KUKA KRL program: Milling_7_1.src

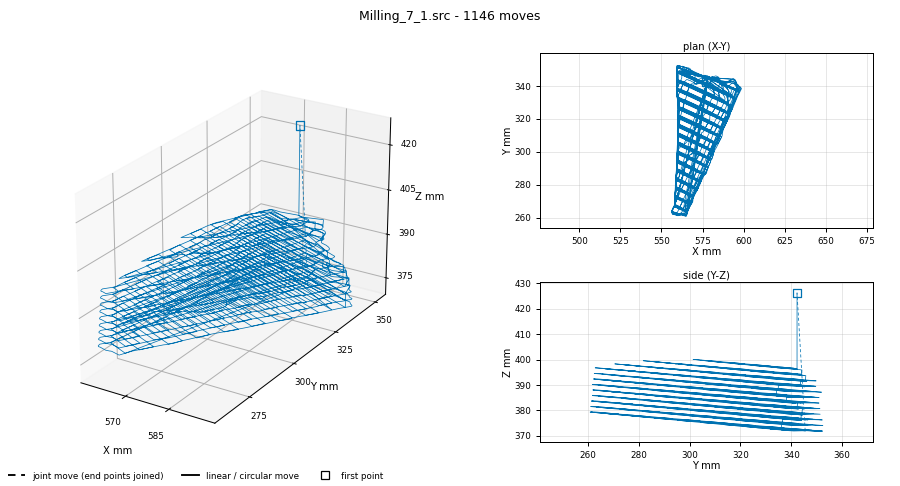
[picture p0: tool path of Milling_7_1.src, 1146 of 1148 moves have a stored position in this frame; points joined in program order, loops and branches not executed]
&ACCESS RVP
&REL 1
&PARAM TEMPLATE = C:\KRC\Roboter\Template\vorgabe
&PARAM EDITMASK = *
DEF Milling_7_1 ( )


;FOLD INI
;FOLD BASISTECH INI
GLOBAL INTERRUPT DECL 3 WHEN $STOPMESS==TRUE DO IR_STOPM ( )
INTERRUPT ON 3
BAS (#INITMOV,0 )
;ENDFOLD (BASISTECH INI)
;ENDFOLD (INI)

;FOLD STARTPOSITION - BASE IS 0, TOOL IS 5, SPEED IS 15%, POSITION IS A1 5,A2 -90,A3 100,A4 5,A5 -10,A6 -5,E1 0,E2 0,E3 0,E4 0
$BWDSTART = FALSE
PDAT_ACT = {VEL 15,ACC 100,APO_DIST 50}
FDAT_ACT = {TOOL_NO 5,BASE_NO 0,IPO_FRAME #BASE}
BAS (#PTP_PARAMS,15)
PTP  {A1 5,A2 -90,A3 100,A4 5,A5 -10,A6 -5,E1 0,E2 0,E3 0,E4 0}
;ENDFOLD

;FOLD LIN SPEED IS 0.1 m/sec, INTERPOLATION SETTINGS IN FOLD
$VEL.CP=0.1
$ADVANCE=3
;ENDFOLD

;FOLD COMMANDS IN FOLD. SELECT EDIT/FOLDS/OPEN ALL FOLDS TO DISPLAY
BAS(#VEL_PTP,2)
PTP {X 576.895, Y 342.279, Z 426.279, A -106.87, B 85.042, C -82.235, E1 0, E2 0, E3 0, E4 0, S 'B010'}
$VEL.CP=0.012
LIN {X 576.895, Y 342.279, Z 396.279, A -106.87, B 85.042, C -82.235, E1 0, E2 0, E3 0, E4 0}
LIN {X 581.744, Y 340.059, Z 396.341, A -106.87, B 85.042, C -82.235, E1 0, E2 0, E3 0, E4 0}
LIN {X 582.117, Y 334.409, Z 396.8, A -106.87, B 85.042, C -82.235, E1 0, E2 0, E3 0, E4 0}
LIN {X 567.684, Y 341.018, Z 396.615, A -106.87, B 85.042, C -82.235, E1 0, E2 0, E3 0, E4 0}
LIN {X 565.563, Y 336.511, Z 397.043, A -106.87, B 85.042, C -82.235, E1 0, E2 0, E3 0, E4 0}
LIN {X 579.527, Y 330.116, Z 397.222, A -106.87, B 85.042, C -82.235, E1 0, E2 0, E3 0, E4 0}
LIN {X 577.52, Y 325.556, Z 397.651, A -106.87, B 85.042, C -82.235, E1 0, E2 0, E3 0, E4 0}
LIN {X 563.782, Y 331.847, Z 397.475, A -106.87, B 85.042, C -82.235, E1 0, E2 0, E3 0, E4 0}
LIN {X 563.044, Y 326.706, Z 397.92, A -106.87, B 85.042, C -82.235, E1 0, E2 0, E3 0, E4 0}
LIN {X 574.933, Y 321.262, Z 398.073, A -106.87, B 85.042, C -82.235, E1 0, E2 0, E3 0, E4 0}
LIN {X 572.822, Y 316.749, Z 398.501, A -106.87, B 85.042, C -82.235, E1 0, E2 0, E3 0, E4 0}
LIN {X 561.971, Y 321.718, Z 398.361, A -106.87, B 85.042, C -82.235, E1 0, E2 0, E3 0, E4 0}
LIN {X 560.617, Y 316.859, Z 398.799, A -106.87, B 85.042, C -82.235, E1 0, E2 0, E3 0, E4 0}
LIN {X 570.047, Y 312.541, Z 398.92, A -106.87, B 85.042, C -82.235, E1 0, E2 0, E3 0, E4 0}
LIN {X 567.602, Y 308.181, Z 399.343, A -106.87, B 85.042, C -82.235, E1 0, E2 0, E3 0, E4 0}
LIN {X 560.515, Y 311.427, Z 399.252, A -106.87, B 85.042, C -82.235, E1 0, E2 0, E3 0, E4 0}
LIN {X 560.232, Y 306.077, Z 399.704, A -106.87, B 85.042, C -82.235, E1 0, E2 0, E3 0, E4 0}
LIN {X 563.648, Y 304.513, Z 399.747, A -106.87, B 85.042, C -82.235, E1 0, E2 0, E3 0, E4 0}
LIN {X 578.662, Y 341.831, Z 396.271, A -106.87, B 85.042, C -82.235, E1 0, E2 0, E3 0, E4 0}
LIN {X 576.305, Y 342.332, Z 396.289, A -106.87, B 85.042, C -82.235, E1 0, E2 0, E3 0, E4 0}
LIN {X 571.991, Y 341.308, Z 396.483, A -106.87, B 85.042, C -82.235, E1 0, E2 0, E3 0, E4 0}
LIN {X 570.835, Y 341.133, Z 396.526, A -106.87, B 85.042, C -82.235, E1 0, E2 0, E3 0, E4 0}
LIN {X 568.535, Y 341.335, Z 396.567, A -106.87, B 85.042, C -82.235, E1 0, E2 0, E3 0, E4 0}
LIN {X 567.853, Y 341.191, Z 396.597, A -106.87, B 85.042, C -82.235, E1 0, E2 0, E3 0, E4 0}
LIN {X 567.158, Y 340.508, Z 396.671, A -106.87, B 85.042, C -82.235, E1 0, E2 0, E3 0, E4 0}
LIN {X 563.05, Y 326.75, Z 397.916, A -106.87, B 85.042, C -82.235, E1 0, E2 0, E3 0, E4 0}
LIN {X 560.877, Y 319.29, Z 398.59, A -106.87, B 85.042, C -82.235, E1 0, E2 0, E3 0, E4 0}
LIN {X 560.632, Y 316.448, Z 398.832, A -106.87, B 85.042, C -82.235, E1 0, E2 0, E3 0, E4 0}
LIN {X 560.608, Y 316.404, Z 398.837, A -106.87, B 85.042, C -82.235, E1 0, E2 0, E3 0, E4 0}
LIN {X 560.617, Y 316.329, Z 398.843, A -106.87, B 85.042, C -82.235, E1 0, E2 0, E3 0, E4 0}
LIN {X 560.448, Y 315.956, Z 398.878, A -106.87, B 85.042, C -82.235, E1 0, E2 0, E3 0, E4 0}
LIN {X 560.332, Y 308.805, Z 399.475, A -106.87, B 85.042, C -82.235, E1 0, E2 0, E3 0, E4 0}
LIN {X 559.954, Y 301.605, Z 400.082, A -106.87, B 85.042, C -82.235, E1 0, E2 0, E3 0, E4 0}
LIN {X 559.952, Y 301.317, Z 400.106, A -106.87, B 85.042, C -82.235, E1 0, E2 0, E3 0, E4 0}
LIN {X 561.639, Y 303.062, Z 399.918, A -106.87, B 85.042, C -82.235, E1 0, E2 0, E3 0, E4 0}
LIN {X 561.767, Y 303.415, Z 399.886, A -106.87, B 85.042, C -82.235, E1 0, E2 0, E3 0, E4 0}
LIN {X 564.546, Y 305.063, Z 399.679, A -106.87, B 85.042, C -82.235, E1 0, E2 0, E3 0, E4 0}
LIN {X 566.478, Y 307.418, Z 399.435, A -106.87, B 85.042, C -82.235, E1 0, E2 0, E3 0, E4 0}
LIN {X 567.57, Y 308.14, Z 399.348, A -106.87, B 85.042, C -82.235, E1 0, E2 0, E3 0, E4 0}
LIN {X 574.106, Y 319.807, Z 398.214, A -106.87, B 85.042, C -82.235, E1 0, E2 0, E3 0, E4 0}
LIN {X 577.01, Y 324.074, Z 397.787, A -106.87, B 85.042, C -82.235, E1 0, E2 0, E3 0, E4 0}
LIN {X 577.887, Y 326.646, Z 397.551, A -106.87, B 85.042, C -82.235, E1 0, E2 0, E3 0, E4 0}
LIN {X 577.83, Y 327.569, Z 397.476, A -106.87, B 85.042, C -82.235, E1 0, E2 0, E3 0, E4 0}
LIN {X 578.067, Y 327.791, Z 397.452, A -106.87, B 85.042, C -82.235, E1 0, E2 0, E3 0, E4 0}
LIN {X 578.437, Y 328.851, Z 397.354, A -106.87, B 85.042, C -82.235, E1 0, E2 0, E3 0, E4 0}
LIN {X 579.308, Y 329.694, Z 397.263, A -106.87, B 85.042, C -82.235, E1 0, E2 0, E3 0, E4 0}
LIN {X 580.616, Y 332.368, Z 397.008, A -106.87, B 85.042, C -82.235, E1 0, E2 0, E3 0, E4 0}
LIN {X 581.829, Y 333.598, Z 396.875, A -106.87, B 85.042, C -82.235, E1 0, E2 0, E3 0, E4 0}
LIN {X 582.26, Y 335.087, Z 396.74, A -106.87, B 85.042, C -82.235, E1 0, E2 0, E3 0, E4 0}
LIN {X 581.267, Y 338.076, Z 396.517, A -106.87, B 85.042, C -82.235, E1 0, E2 0, E3 0, E4 0}
LIN {X 581.747, Y 340.003, Z 396.345, A -106.87, B 85.042, C -82.235, E1 0, E2 0, E3 0, E4 0}
LIN {X 581.733, Y 340.279, Z 396.323, A -106.87, B 85.042, C -82.235, E1 0, E2 0, E3 0, E4 0}
LIN {X 580.797, Y 341.376, Z 396.255, A -106.87, B 85.042, C -82.235, E1 0, E2 0, E3 0, E4 0}
LIN {X 578.662, Y 341.831, Z 396.271, A -106.87, B 85.042, C -82.235, E1 0, E2 0, E3 0, E4 0}
LIN {X 584.625, Y 344.218, Z 395.923, A -106.87, B 85.042, C -82.235, E1 0, E2 0, E3 0, E4 0}
LIN {X 584.571, Y 344.039, Z 393.757, A -106.87, B 85.042, C -82.235, E1 0, E2 0, E3 0, E4 0}
LIN {X 582.705, Y 344.893, Z 393.733, A -106.87, B 85.042, C -82.235, E1 0, E2 0, E3 0, E4 0}
LIN {X 574.324, Y 343.252, Z 394.08, A -106.87, B 85.042, C -82.235, E1 0, E2 0, E3 0, E4 0}
LIN {X 584.3, Y 338.684, Z 394.209, A -106.87, B 85.042, C -82.235, E1 0, E2 0, E3 0, E4 0}
LIN {X 585.153, Y 332.814, Z 394.674, A -106.87, B 85.042, C -82.235, E1 0, E2 0, E3 0, E4 0}
LIN {X 563.874, Y 342.559, Z 394.401, A -106.87, B 85.042, C -82.235, E1 0, E2 0, E3 0, E4 0}
LIN {X 561.643, Y 338.101, Z 394.827, A -106.87, B 85.042, C -82.235, E1 0, E2 0, E3 0, E4 0}
LIN {X 583.515, Y 328.084, Z 395.108, A -106.87, B 85.042, C -82.235, E1 0, E2 0, E3 0, E4 0}
LIN {X 580.918, Y 323.795, Z 395.53, A -106.87, B 85.042, C -82.235, E1 0, E2 0, E3 0, E4 0}
LIN {X 560.439, Y 333.174, Z 395.267, A -106.87, B 85.042, C -82.235, E1 0, E2 0, E3 0, E4 0}
LIN {X 560.554, Y 327.641, Z 395.723, A -106.87, B 85.042, C -82.235, E1 0, E2 0, E3 0, E4 0}
LIN {X 579.074, Y 319.16, Z 395.961, A -106.87, B 85.042, C -82.235, E1 0, E2 0, E3 0, E4 0}
LIN {X 576.813, Y 314.717, Z 396.387, A -106.87, B 85.042, C -82.235, E1 0, E2 0, E3 0, E4 0}
LIN {X 560.377, Y 322.243, Z 396.176, A -106.87, B 85.042, C -82.235, E1 0, E2 0, E3 0, E4 0}
LIN {X 560.494, Y 316.71, Z 396.632, A -106.87, B 85.042, C -82.235, E1 0, E2 0, E3 0, E4 0}
LIN {X 574.212, Y 310.428, Z 396.808, A -106.87, B 85.042, C -82.235, E1 0, E2 0, E3 0, E4 0}
LIN {X 572.498, Y 305.734, Z 397.241, A -106.87, B 85.042, C -82.235, E1 0, E2 0, E3 0, E4 0}
LIN {X 560.46, Y 311.247, Z 397.087, A -106.87, B 85.042, C -82.235, E1 0, E2 0, E3 0, E4 0}
LIN {X 560.177, Y 305.898, Z 397.538, A -106.87, B 85.042, C -82.235, E1 0, E2 0, E3 0, E4 0}
LIN {X 570.719, Y 301.07, Z 397.673, A -106.87, B 85.042, C -82.235, E1 0, E2 0, E3 0, E4 0}
LIN {X 566.667, Y 297.446, Z 398.076, A -106.87, B 85.042, C -82.235, E1 0, E2 0, E3 0, E4 0}
LIN {X 559.925, Y 300.534, Z 397.989, A -106.87, B 85.042, C -82.235, E1 0, E2 0, E3 0, E4 0}
LIN {X 560.131, Y 294.96, Z 398.447, A -106.87, B 85.042, C -82.235, E1 0, E2 0, E3 0, E4 0}
LIN {X 563.737, Y 293.309, Z 398.493, A -106.87, B 85.042, C -82.235, E1 0, E2 0, E3 0, E4 0}
LIN {X 562.482, Y 288.404, Z 398.932, A -106.87, B 85.042, C -82.235, E1 0, E2 0, E3 0, E4 0}
LIN {X 559.719, Y 289.67, Z 398.896, A -106.87, B 85.042, C -82.235, E1 0, E2 0, E3 0, E4 0}
LIN {X 559.06, Y 284.492, Z 399.343, A -106.87, B 85.042, C -82.235, E1 0, E2 0, E3 0, E4 0}
LIN {X 560.33, Y 283.911, Z 399.359, A -106.87, B 85.042, C -82.235, E1 0, E2 0, E3 0, E4 0}
LIN {X 578.097, Y 344.003, Z 393.923, A -106.87, B 85.042, C -82.235, E1 0, E2 0, E3 0, E4 0}
LIN {X 583.583, Y 345.174, Z 393.688, A -106.87, B 85.042, C -82.235, E1 0, E2 0, E3 0, E4 0}
LIN {X 583.658, Y 345.166, Z 393.687, A -106.87, B 85.042, C -82.235, E1 0, E2 0, E3 0, E4 0}
LIN {X 583.724, Y 345.117, Z 393.689, A -106.87, B 85.042, C -82.235, E1 0, E2 0, E3 0, E4 0}
LIN {X 585.069, Y 343.343, Z 393.802, A -106.87, B 85.042, C -82.235, E1 0, E2 0, E3 0, E4 0}
LIN {X 585.534, Y 341.633, Z 393.933, A -106.87, B 85.042, C -82.235, E1 0, E2 0, E3 0, E4 0}
LIN {X 585.454, Y 341.123, Z 393.977, A -106.87, B 85.042, C -82.235, E1 0, E2 0, E3 0, E4 0}
LIN {X 584.65, Y 339.762, Z 394.11, A -106.87, B 85.042, C -82.235, E1 0, E2 0, E3 0, E4 0}
LIN {X 584.558, Y 339.684, Z 394.119, A -106.87, B 85.042, C -82.235, E1 0, E2 0, E3 0, E4 0}
LIN {X 584.115, Y 337.478, Z 394.313, A -106.87, B 85.042, C -82.235, E1 0, E2 0, E3 0, E4 0}
LIN {X 585.114, Y 335.114, Z 394.484, A -106.87, B 85.042, C -82.235, E1 0, E2 0, E3 0, E4 0}
LIN {X 585.144, Y 332.703, Z 394.684, A -106.87, B 85.042, C -82.235, E1 0, E2 0, E3 0, E4 0}
LIN {X 584.551, Y 331.291, Z 394.816, A -106.87, B 85.042, C -82.235, E1 0, E2 0, E3 0, E4 0}
LIN {X 584.057, Y 330.694, Z 394.878, A -106.87, B 85.042, C -82.235, E1 0, E2 0, E3 0, E4 0}
LIN {X 583.581, Y 328.244, Z 395.093, A -106.87, B 85.042, C -82.235, E1 0, E2 0, E3 0, E4 0}
LIN {X 580.825, Y 323.667, Z 395.543, A -106.87, B 85.042, C -82.235, E1 0, E2 0, E3 0, E4 0}
LIN {X 579.822, Y 323.235, Z 395.604, A -106.87, B 85.042, C -82.235, E1 0, E2 0, E3 0, E4 0}
LIN {X 579.732, Y 323.124, Z 395.615, A -106.87, B 85.042, C -82.235, E1 0, E2 0, E3 0, E4 0}
LIN {X 579.441, Y 322.375, Z 395.685, A -106.87, B 85.042, C -82.235, E1 0, E2 0, E3 0, E4 0}
LIN {X 579.352, Y 319.987, Z 395.885, A -106.87, B 85.042, C -82.235, E1 0, E2 0, E3 0, E4 0}
LIN {X 576.924, Y 315.102, Z 396.352, A -106.87, B 85.042, C -82.235, E1 0, E2 0, E3 0, E4 0}
LIN {X 576.416, Y 313.428, Z 396.504, A -106.87, B 85.042, C -82.235, E1 0, E2 0, E3 0, E4 0}
LIN {X 575.142, Y 311.958, Z 396.658, A -106.87, B 85.042, C -82.235, E1 0, E2 0, E3 0, E4 0}
LIN {X 574.554, Y 311.675, Z 396.696, A -106.87, B 85.042, C -82.235, E1 0, E2 0, E3 0, E4 0}
LIN {X 574.252, Y 311.233, Z 396.74, A -106.87, B 85.042, C -82.235, E1 0, E2 0, E3 0, E4 0}
LIN {X 574.21, Y 309.999, Z 396.844, A -106.87, B 85.042, C -82.235, E1 0, E2 0, E3 0, E4 0}
LIN {X 570.659, Y 300.834, Z 397.694, A -106.87, B 85.042, C -82.235, E1 0, E2 0, E3 0, E4 0}
LIN {X 569.22, Y 298.941, Z 397.888, A -106.87, B 85.042, C -82.235, E1 0, E2 0, E3 0, E4 0}
LIN {X 566.753, Y 297.93, Z 398.034, A -106.87, B 85.042, C -82.235, E1 0, E2 0, E3 0, E4 0}
LIN {X 566.692, Y 297.837, Z 398.043, A -106.87, B 85.042, C -82.235, E1 0, E2 0, E3 0, E4 0}
LIN {X 566.762, Y 296.23, Z 398.175, A -106.87, B 85.042, C -82.235, E1 0, E2 0, E3 0, E4 0}
LIN {X 566.431, Y 295.493, Z 398.244, A -106.87, B 85.042, C -82.235, E1 0, E2 0, E3 0, E4 0}
LIN {X 566.28, Y 294.839, Z 398.302, A -106.87, B 85.042, C -82.235, E1 0, E2 0, E3 0, E4 0}
LIN {X 565.783, Y 294.409, Z 398.35, A -106.87, B 85.042, C -82.235, E1 0, E2 0, E3 0, E4 0}
LIN {X 565.156, Y 294.696, Z 398.342, A -106.87, B 85.042, C -82.235, E1 0, E2 0, E3 0, E4 0}
LIN {X 564.945, Y 294.236, Z 398.386, A -106.87, B 85.042, C -82.235, E1 0, E2 0, E3 0, E4 0}
LIN {X 564.12, Y 293.972, Z 398.429, A -106.87, B 85.042, C -82.235, E1 0, E2 0, E3 0, E4 0}
LIN {X 563.85, Y 293.432, Z 398.48, A -106.87, B 85.042, C -82.235, E1 0, E2 0, E3 0, E4 0}
LIN {X 563.685, Y 293.251, Z 398.499, A -106.87, B 85.042, C -82.235, E1 0, E2 0, E3 0, E4 0}
LIN {X 564.591, Y 292.757, Z 398.518, A -106.87, B 85.042, C -82.235, E1 0, E2 0, E3 0, E4 0}
LIN {X 564.637, Y 292.748, Z 398.517, A -106.87, B 85.042, C -82.235, E1 0, E2 0, E3 0, E4 0}
LIN {X 564.633, Y 292.727, Z 398.519, A -106.87, B 85.042, C -82.235, E1 0, E2 0, E3 0, E4 0}
LIN {X 564.76, Y 291.881, Z 398.586, A -106.87, B 85.042, C -82.235, E1 0, E2 0, E3 0, E4 0}
LIN {X 564.136, Y 290.632, Z 398.705, A -106.87, B 85.042, C -82.235, E1 0, E2 0, E3 0, E4 0}
LIN {X 563.633, Y 290.496, Z 398.729, A -106.87, B 85.042, C -82.235, E1 0, E2 0, E3 0, E4 0}
LIN {X 563.816, Y 290.033, Z 398.763, A -106.87, B 85.042, C -82.235, E1 0, E2 0, E3 0, E4 0}
LIN {X 562.653, Y 288.496, Z 398.92, A -106.87, B 85.042, C -82.235, E1 0, E2 0, E3 0, E4 0}
LIN {X 562.089, Y 288.191, Z 398.96, A -106.87, B 85.042, C -82.235, E1 0, E2 0, E3 0, E4 0}
LIN {X 561.588, Y 287.183, Z 399.056, A -106.87, B 85.042, C -82.235, E1 0, E2 0, E3 0, E4 0}
LIN {X 561.726, Y 286.954, Z 399.071, A -106.87, B 85.042, C -82.235, E1 0, E2 0, E3 0, E4 0}
LIN {X 561.239, Y 286.678, Z 399.107, A -106.87, B 85.042, C -82.235, E1 0, E2 0, E3 0, E4 0}
LIN {X 561.257, Y 286.467, Z 399.124, A -106.87, B 85.042, C -82.235, E1 0, E2 0, E3 0, E4 0}
LIN {X 560.71, Y 284.65, Z 399.288, A -106.87, B 85.042, C -82.235, E1 0, E2 0, E3 0, E4 0}
LIN {X 559.03, Y 281.698, Z 399.576, A -106.87, B 85.042, C -82.235, E1 0, E2 0, E3 0, E4 0}
LIN {X 560.519, Y 309.67, Z 397.216, A -106.87, B 85.042, C -82.235, E1 0, E2 0, E3 0, E4 0}
LIN {X 560.165, Y 314.552, Z 396.82, A -106.87, B 85.042, C -82.235, E1 0, E2 0, E3 0, E4 0}
LIN {X 560.562, Y 316.149, Z 396.677, A -106.87, B 85.042, C -82.235, E1 0, E2 0, E3 0, E4 0}
LIN {X 560.48, Y 317.178, Z 396.594, A -106.87, B 85.042, C -82.235, E1 0, E2 0, E3 0, E4 0}
LIN {X 560.446, Y 317.247, Z 396.589, A -106.87, B 85.042, C -82.235, E1 0, E2 0, E3 0, E4 0}
LIN {X 560.814, Y 330.69, Z 395.464, A -106.87, B 85.042, C -82.235, E1 0, E2 0, E3 0, E4 0}
LIN {X 560.738, Y 330.851, Z 395.452, A -106.87, B 85.042, C -82.235, E1 0, E2 0, E3 0, E4 0}
LIN {X 560.306, Y 334.39, Z 395.169, A -106.87, B 85.042, C -82.235, E1 0, E2 0, E3 0, E4 0}
LIN {X 563.334, Y 341.786, Z 394.479, A -106.87, B 85.042, C -82.235, E1 0, E2 0, E3 0, E4 0}
LIN {X 565.199, Y 343.887, Z 394.257, A -106.87, B 85.042, C -82.235, E1 0, E2 0, E3 0, E4 0}
LIN {X 566.09, Y 343.841, Z 394.239, A -106.87, B 85.042, C -82.235, E1 0, E2 0, E3 0, E4 0}
LIN {X 566.53, Y 343.532, Z 394.253, A -106.87, B 85.042, C -82.235, E1 0, E2 0, E3 0, E4 0}
LIN {X 567.45, Y 343.318, Z 394.248, A -106.87, B 85.042, C -82.235, E1 0, E2 0, E3 0, E4 0}
LIN {X 570.821, Y 341.414, Z 394.321, A -106.87, B 85.042, C -82.235, E1 0, E2 0, E3 0, E4 0}
LIN {X 571.518, Y 341.33, Z 394.311, A -106.87, B 85.042, C -82.235, E1 0, E2 0, E3 0, E4 0}
LIN {X 573.337, Y 342.631, Z 394.157, A -106.87, B 85.042, C -82.235, E1 0, E2 0, E3 0, E4 0}
LIN {X 573.683, Y 343.06, Z 394.112, A -106.87, B 85.042, C -82.235, E1 0, E2 0, E3 0, E4 0}
LIN {X 578.097, Y 344.003, Z 393.923, A -106.87, B 85.042, C -82.235, E1 0, E2 0, E3 0, E4 0}
LIN {X 580.876, Y 345.731, Z 393.71, A -106.87, B 85.042, C -82.235, E1 0, E2 0, E3 0, E4 0}
LIN {X 580.822, Y 345.551, Z 391.544, A -106.87, B 85.042, C -82.235, E1 0, E2 0, E3 0, E4 0}
LIN {X 585.842, Y 343.252, Z 391.608, A -106.87, B 85.042, C -82.235, E1 0, E2 0, E3 0, E4 0}
LIN {X 587.33, Y 337.091, Z 392.082, A -106.87, B 85.042, C -82.235, E1 0, E2 0, E3 0, E4 0}
LIN {X 572.399, Y 343.929, Z 391.891, A -106.87, B 85.042, C -82.235, E1 0, E2 0, E3 0, E4 0}
LIN {X 562.627, Y 348.404, Z 391.765, A -106.87, B 85.042, C -82.235, E1 0, E2 0, E3 0, E4 0}
LIN {X 570.487, Y 344.804, Z 391.866, A -106.87, B 85.042, C -82.235, E1 0, E2 0, E3 0, E4 0}
LIN {X 588.468, Y 331.091, Z 392.552, A -106.87, B 85.042, C -82.235, E1 0, E2 0, E3 0, E4 0}
LIN {X 561.576, Y 343.406, Z 392.207, A -106.87, B 85.042, C -82.235, E1 0, E2 0, E3 0, E4 0}
LIN {X 559.643, Y 338.812, Z 392.637, A -106.87, B 85.042, C -82.235, E1 0, E2 0, E3 0, E4 0}
LIN {X 586.399, Y 326.559, Z 392.98, A -106.87, B 85.042, C -82.235, E1 0, E2 0, E3 0, E4 0}
LIN {X 584.074, Y 322.145, Z 393.405, A -106.87, B 85.042, C -82.235, E1 0, E2 0, E3 0, E4 0}
LIN {X 560.384, Y 332.994, Z 393.101, A -106.87, B 85.042, C -82.235, E1 0, E2 0, E3 0, E4 0}
LIN {X 560.5, Y 327.462, Z 393.557, A -106.87, B 85.042, C -82.235, E1 0, E2 0, E3 0, E4 0}
LIN {X 581.809, Y 317.703, Z 393.831, A -106.87, B 85.042, C -82.235, E1 0, E2 0, E3 0, E4 0}
LIN {X 579.849, Y 313.121, Z 394.261, A -106.87, B 85.042, C -82.235, E1 0, E2 0, E3 0, E4 0}
LIN {X 560.323, Y 322.063, Z 394.01, A -106.87, B 85.042, C -82.235, E1 0, E2 0, E3 0, E4 0}
LIN {X 560.44, Y 316.531, Z 394.466, A -106.87, B 85.042, C -82.235, E1 0, E2 0, E3 0, E4 0}
LIN {X 577.836, Y 308.564, Z 394.69, A -106.87, B 85.042, C -82.235, E1 0, E2 0, E3 0, E4 0}
LIN {X 575.845, Y 303.996, Z 395.119, A -106.87, B 85.042, C -82.235, E1 0, E2 0, E3 0, E4 0}
LIN {X 560.406, Y 311.067, Z 394.921, A -106.87, B 85.042, C -82.235, E1 0, E2 0, E3 0, E4 0}
LIN {X 560.122, Y 305.718, Z 395.372, A -106.87, B 85.042, C -82.235, E1 0, E2 0, E3 0, E4 0}
LIN {X 573.777, Y 299.464, Z 395.547, A -106.87, B 85.042, C -82.235, E1 0, E2 0, E3 0, E4 0}
LIN {X 571.315, Y 295.113, Z 395.971, A -106.87, B 85.042, C -82.235, E1 0, E2 0, E3 0, E4 0}
LIN {X 559.871, Y 300.354, Z 395.824, A -106.87, B 85.042, C -82.235, E1 0, E2 0, E3 0, E4 0}
LIN {X 560.076, Y 294.781, Z 396.281, A -106.87, B 85.042, C -82.235, E1 0, E2 0, E3 0, E4 0}
LIN {X 569.346, Y 290.535, Z 396.4, A -106.87, B 85.042, C -82.235, E1 0, E2 0, E3 0, E4 0}
LIN {X 566.96, Y 286.149, Z 396.824, A -106.87, B 85.042, C -82.235, E1 0, E2 0, E3 0, E4 0}
LIN {X 559.664, Y 289.49, Z 396.731, A -106.87, B 85.042, C -82.235, E1 0, E2 0, E3 0, E4 0}
LIN {X 559.006, Y 284.312, Z 397.177, A -106.87, B 85.042, C -82.235, E1 0, E2 0, E3 0, E4 0}
LIN {X 564.493, Y 281.799, Z 397.248, A -106.87, B 85.042, C -82.235, E1 0, E2 0, E3 0, E4 0}
LIN {X 562.21, Y 277.366, Z 397.673, A -106.87, B 85.042, C -82.235, E1 0, E2 0, E3 0, E4 0}
LIN {X 558.844, Y 278.907, Z 397.63, A -106.87, B 85.042, C -82.235, E1 0, E2 0, E3 0, E4 0}
LIN {X 558.518, Y 273.577, Z 398.081, A -106.87, B 85.042, C -82.235, E1 0, E2 0, E3 0, E4 0}
LIN {X 559.993, Y 272.902, Z 398.1, A -106.87, B 85.042, C -82.235, E1 0, E2 0, E3 0, E4 0}
LIN {X 578.218, Y 345.098, Z 391.647, A -106.87, B 85.042, C -82.235, E1 0, E2 0, E3 0, E4 0}
LIN {X 579.101, Y 344.975, Z 391.635, A -106.87, B 85.042, C -82.235, E1 0, E2 0, E3 0, E4 0}
LIN {X 583.083, Y 346.167, Z 391.436, A -106.87, B 85.042, C -82.235, E1 0, E2 0, E3 0, E4 0}
LIN {X 584.478, Y 345.556, Z 391.451, A -106.87, B 85.042, C -82.235, E1 0, E2 0, E3 0, E4 0}
LIN {X 585.511, Y 344.183, Z 391.539, A -106.87, B 85.042, C -82.235, E1 0, E2 0, E3 0, E4 0}
LIN {X 586.277, Y 340.991, Z 391.785, A -106.87, B 85.042, C -82.235, E1 0, E2 0, E3 0, E4 0}
LIN {X 587.074, Y 340.037, Z 391.844, A -106.87, B 85.042, C -82.235, E1 0, E2 0, E3 0, E4 0}
LIN {X 587.651, Y 339.495, Z 391.875, A -106.87, B 85.042, C -82.235, E1 0, E2 0, E3 0, E4 0}
LIN {X 587.856, Y 338.588, Z 391.945, A -106.87, B 85.042, C -82.235, E1 0, E2 0, E3 0, E4 0}
LIN {X 587.296, Y 336.993, Z 392.091, A -106.87, B 85.042, C -82.235, E1 0, E2 0, E3 0, E4 0}
LIN {X 587.229, Y 335.812, Z 392.191, A -106.87, B 85.042, C -82.235, E1 0, E2 0, E3 0, E4 0}
LIN {X 587.483, Y 334.662, Z 392.28, A -106.87, B 85.042, C -82.235, E1 0, E2 0, E3 0, E4 0}
LIN {X 588.142, Y 333.798, Z 392.335, A -106.87, B 85.042, C -82.235, E1 0, E2 0, E3 0, E4 0}
LIN {X 588.645, Y 332.542, Z 392.427, A -106.87, B 85.042, C -82.235, E1 0, E2 0, E3 0, E4 0}
LIN {X 588.395, Y 330.692, Z 392.587, A -106.87, B 85.042, C -82.235, E1 0, E2 0, E3 0, E4 0}
LIN {X 581.012, Y 315.463, Z 394.037, A -106.87, B 85.042, C -82.235, E1 0, E2 0, E3 0, E4 0}
LIN {X 561.669, Y 276.539, Z 397.755, A -106.87, B 85.042, C -82.235, E1 0, E2 0, E3 0, E4 0}
LIN {X 561.673, Y 276.429, Z 397.764, A -106.87, B 85.042, C -82.235, E1 0, E2 0, E3 0, E4 0}
LIN {X 560.774, Y 274.04, Z 397.986, A -106.87, B 85.042, C -82.235, E1 0, E2 0, E3 0, E4 0}
LIN {X 558.721, Y 270.49, Z 398.332, A -106.87, B 85.042, C -82.235, E1 0, E2 0, E3 0, E4 0}
LIN {X 558.537, Y 272.628, Z 398.159, A -106.87, B 85.042, C -82.235, E1 0, E2 0, E3 0, E4 0}
LIN {X 558.828, Y 276.652, Z 397.818, A -106.87, B 85.042, C -82.235, E1 0, E2 0, E3 0, E4 0}
LIN {X 560.465, Y 309.49, Z 395.05, A -106.87, B 85.042, C -82.235, E1 0, E2 0, E3 0, E4 0}
LIN {X 560.11, Y 314.372, Z 394.654, A -106.87, B 85.042, C -82.235, E1 0, E2 0, E3 0, E4 0}
LIN {X 560.508, Y 315.969, Z 394.511, A -106.87, B 85.042, C -82.235, E1 0, E2 0, E3 0, E4 0}
LIN {X 560.425, Y 316.998, Z 394.428, A -106.87, B 85.042, C -82.235, E1 0, E2 0, E3 0, E4 0}
LIN {X 560.391, Y 317.067, Z 394.423, A -106.87, B 85.042, C -82.235, E1 0, E2 0, E3 0, E4 0}
LIN {X 560.759, Y 330.511, Z 393.298, A -106.87, B 85.042, C -82.235, E1 0, E2 0, E3 0, E4 0}
LIN {X 560.683, Y 330.671, Z 393.286, A -106.87, B 85.042, C -82.235, E1 0, E2 0, E3 0, E4 0}
LIN {X 559.737, Y 335.976, Z 392.87, A -106.87, B 85.042, C -82.235, E1 0, E2 0, E3 0, E4 0}
LIN {X 559.647, Y 339.062, Z 392.616, A -106.87, B 85.042, C -82.235, E1 0, E2 0, E3 0, E4 0}
LIN {X 562.296, Y 344.753, Z 392.077, A -106.87, B 85.042, C -82.235, E1 0, E2 0, E3 0, E4 0}
LIN {X 562.552, Y 349.38, Z 391.686, A -106.87, B 85.042, C -82.235, E1 0, E2 0, E3 0, E4 0}
LIN {X 562.628, Y 349.761, Z 391.652, A -106.87, B 85.042, C -82.235, E1 0, E2 0, E3 0, E4 0}
LIN {X 562.694, Y 349.794, Z 391.648, A -106.87, B 85.042, C -82.235, E1 0, E2 0, E3 0, E4 0}
LIN {X 566.596, Y 348.974, Z 391.618, A -106.87, B 85.042, C -82.235, E1 0, E2 0, E3 0, E4 0}
LIN {X 569.925, Y 347.68, Z 391.641, A -106.87, B 85.042, C -82.235, E1 0, E2 0, E3 0, E4 0}
LIN {X 570.226, Y 347.271, Z 391.668, A -106.87, B 85.042, C -82.235, E1 0, E2 0, E3 0, E4 0}
LIN {X 570.209, Y 347.141, Z 391.679, A -106.87, B 85.042, C -82.235, E1 0, E2 0, E3 0, E4 0}
LIN {X 570.438, Y 346.095, Z 391.76, A -106.87, B 85.042, C -82.235, E1 0, E2 0, E3 0, E4 0}
LIN {X 570.351, Y 344.929, Z 391.859, A -106.87, B 85.042, C -82.235, E1 0, E2 0, E3 0, E4 0}
LIN {X 571.715, Y 343.685, Z 391.928, A -106.87, B 85.042, C -82.235, E1 0, E2 0, E3 0, E4 0}
LIN {X 569.859, Y 343.017, Z 392.03, A -106.87, B 85.042, C -82.235, E1 0, E2 0, E3 0, E4 0}
LIN {X 569.861, Y 342.66, Z 392.06, A -106.87, B 85.042, C -82.235, E1 0, E2 0, E3 0, E4 0}
LIN {X 569.65, Y 342.247, Z 392.099, A -106.87, B 85.042, C -82.235, E1 0, E2 0, E3 0, E4 0}
LIN {X 570.082, Y 341.636, Z 392.139, A -106.87, B 85.042, C -82.235, E1 0, E2 0, E3 0, E4 0}
LIN {X 570.349, Y 341.468, Z 392.147, A -106.87, B 85.042, C -82.235, E1 0, E2 0, E3 0, E4 0}
LIN {X 571.203, Y 341.242, Z 392.144, A -106.87, B 85.042, C -82.235, E1 0, E2 0, E3 0, E4 0}
LIN {X 571.783, Y 343.654, Z 391.929, A -106.87, B 85.042, C -82.235, E1 0, E2 0, E3 0, E4 0}
LIN {X 571.795, Y 343.669, Z 391.927, A -106.87, B 85.042, C -82.235, E1 0, E2 0, E3 0, E4 0}
LIN {X 574.195, Y 344.701, Z 391.781, A -106.87, B 85.042, C -82.235, E1 0, E2 0, E3 0, E4 0}
LIN {X 576.649, Y 344.932, Z 391.7, A -106.87, B 85.042, C -82.235, E1 0, E2 0, E3 0, E4 0}
LIN {X 577.654, Y 345.176, Z 391.655, A -106.87, B 85.042, C -82.235, E1 0, E2 0, E3 0, E4 0}
LIN {X 578.218, Y 345.098, Z 391.647, A -106.87, B 85.042, C -82.235, E1 0, E2 0, E3 0, E4 0}
LIN {X 584.892, Y 343.687, Z 391.596, A -106.87, B 85.042, C -82.235, E1 0, E2 0, E3 0, E4 0}
LIN {X 584.837, Y 343.507, Z 389.43, A -106.87, B 85.042, C -82.235, E1 0, E2 0, E3 0, E4 0}
LIN {X 581.654, Y 344.965, Z 389.389, A -106.87, B 85.042, C -82.235, E1 0, E2 0, E3 0, E4 0}
LIN {X 560.751, Y 349.059, Z 389.576, A -106.87, B 85.042, C -82.235, E1 0, E2 0, E3 0, E4 0}
LIN {X 590.147, Y 335.596, Z 389.954, A -106.87, B 85.042, C -82.235, E1 0, E2 0, E3 0, E4 0}
LIN {X 590.276, Y 330.058, Z 390.41, A -106.87, B 85.042, C -82.235, E1 0, E2 0, E3 0, E4 0}
LIN {X 559.646, Y 344.085, Z 390.017, A -106.87, B 85.042, C -82.235, E1 0, E2 0, E3 0, E4 0}
LIN {X 559.589, Y 338.633, Z 390.471, A -106.87, B 85.042, C -82.235, E1 0, E2 0, E3 0, E4 0}
LIN {X 588.617, Y 325.339, Z 390.844, A -106.87, B 85.042, C -82.235, E1 0, E2 0, E3 0, E4 0}
LIN {X 586.307, Y 320.917, Z 391.269, A -106.87, B 85.042, C -82.235, E1 0, E2 0, E3 0, E4 0}
LIN {X 560.33, Y 332.814, Z 390.935, A -106.87, B 85.042, C -82.235, E1 0, E2 0, E3 0, E4 0}
LIN {X 560.445, Y 327.282, Z 391.392, A -106.87, B 85.042, C -82.235, E1 0, E2 0, E3 0, E4 0}
LIN {X 584.357, Y 316.331, Z 391.699, A -106.87, B 85.042, C -82.235, E1 0, E2 0, E3 0, E4 0}
LIN {X 582.293, Y 311.797, Z 392.127, A -106.87, B 85.042, C -82.235, E1 0, E2 0, E3 0, E4 0}
LIN {X 560.268, Y 321.884, Z 391.844, A -106.87, B 85.042, C -82.235, E1 0, E2 0, E3 0, E4 0}
LIN {X 560.385, Y 316.351, Z 392.301, A -106.87, B 85.042, C -82.235, E1 0, E2 0, E3 0, E4 0}
LIN {X 580.214, Y 307.27, Z 392.555, A -106.87, B 85.042, C -82.235, E1 0, E2 0, E3 0, E4 0}
LIN {X 578.281, Y 302.676, Z 392.985, A -106.87, B 85.042, C -82.235, E1 0, E2 0, E3 0, E4 0}
LIN {X 560.351, Y 310.887, Z 392.755, A -106.87, B 85.042, C -82.235, E1 0, E2 0, E3 0, E4 0}
LIN {X 560.068, Y 305.538, Z 393.206, A -106.87, B 85.042, C -82.235, E1 0, E2 0, E3 0, E4 0}
LIN {X 576.165, Y 298.166, Z 393.413, A -106.87, B 85.042, C -82.235, E1 0, E2 0, E3 0, E4 0}
LIN {X 574.194, Y 293.59, Z 393.842, A -106.87, B 85.042, C -82.235, E1 0, E2 0, E3 0, E4 0}
LIN {X 559.816, Y 300.174, Z 393.658, A -106.87, B 85.042, C -82.235, E1 0, E2 0, E3 0, E4 0}
LIN {X 560.022, Y 294.601, Z 394.115, A -106.87, B 85.042, C -82.235, E1 0, E2 0, E3 0, E4 0}
LIN {X 572.043, Y 289.096, Z 394.27, A -106.87, B 85.042, C -82.235, E1 0, E2 0, E3 0, E4 0}
LIN {X 569.847, Y 284.622, Z 394.696, A -106.87, B 85.042, C -82.235, E1 0, E2 0, E3 0, E4 0}
LIN {X 559.609, Y 289.31, Z 394.565, A -106.87, B 85.042, C -82.235, E1 0, E2 0, E3 0, E4 0}
LIN {X 558.951, Y 284.133, Z 395.011, A -106.87, B 85.042, C -82.235, E1 0, E2 0, E3 0, E4 0}
LIN {X 568.041, Y 279.97, Z 395.128, A -106.87, B 85.042, C -82.235, E1 0, E2 0, E3 0, E4 0}
LIN {X 565.556, Y 275.628, Z 395.551, A -106.87, B 85.042, C -82.235, E1 0, E2 0, E3 0, E4 0}
LIN {X 558.789, Y 278.728, Z 395.464, A -106.87, B 85.042, C -82.235, E1 0, E2 0, E3 0, E4 0}
LIN {X 558.463, Y 273.398, Z 395.915, A -106.87, B 85.042, C -82.235, E1 0, E2 0, E3 0, E4 0}
LIN {X 563.541, Y 271.072, Z 395.98, A -106.87, B 85.042, C -82.235, E1 0, E2 0, E3 0, E4 0}
LIN {X 561.262, Y 266.637, Z 396.406, A -106.87, B 85.042, C -82.235, E1 0, E2 0, E3 0, E4 0}
LIN {X 558.324, Y 267.982, Z 396.368, A -106.87, B 85.042, C -82.235, E1 0, E2 0, E3 0, E4 0}
LIN {X 578.154, Y 344.821, Z 389.49, A -106.87, B 85.042, C -82.235, E1 0, E2 0, E3 0, E4 0}
LIN {X 580.331, Y 344.607, Z 389.453, A -106.87, B 85.042, C -82.235, E1 0, E2 0, E3 0, E4 0}
LIN {X 583.657, Y 345.363, Z 389.306, A -106.87, B 85.042, C -82.235, E1 0, E2 0, E3 0, E4 0}
LIN {X 584.034, Y 345.169, Z 389.313, A -106.87, B 85.042, C -82.235, E1 0, E2 0, E3 0, E4 0}
LIN {X 585.184, Y 342.399, Z 389.514, A -106.87, B 85.042, C -82.235, E1 0, E2 0, E3 0, E4 0}
LIN {X 585.762, Y 341.122, Z 389.605, A -106.87, B 85.042, C -82.235, E1 0, E2 0, E3 0, E4 0}
LIN {X 586.211, Y 340.748, Z 389.625, A -106.87, B 85.042, C -82.235, E1 0, E2 0, E3 0, E4 0}
LIN {X 588.162, Y 340.013, Z 389.637, A -106.87, B 85.042, C -82.235, E1 0, E2 0, E3 0, E4 0}
LIN {X 589.656, Y 338.99, Z 389.684, A -106.87, B 85.042, C -82.235, E1 0, E2 0, E3 0, E4 0}
LIN {X 590.535, Y 337.925, Z 389.75, A -106.87, B 85.042, C -82.235, E1 0, E2 0, E3 0, E4 0}
LIN {X 590.85, Y 336.932, Z 389.825, A -106.87, B 85.042, C -82.235, E1 0, E2 0, E3 0, E4 0}
LIN {X 590.748, Y 336.368, Z 389.874, A -106.87, B 85.042, C -82.235, E1 0, E2 0, E3 0, E4 0}
LIN {X 590.588, Y 336.043, Z 389.905, A -106.87, B 85.042, C -82.235, E1 0, E2 0, E3 0, E4 0}
LIN {X 589.712, Y 335.082, Z 390.007, A -106.87, B 85.042, C -82.235, E1 0, E2 0, E3 0, E4 0}
LIN {X 589.573, Y 333.596, Z 390.134, A -106.87, B 85.042, C -82.235, E1 0, E2 0, E3 0, E4 0}
LIN {X 590.534, Y 331.255, Z 390.304, A -106.87, B 85.042, C -82.235, E1 0, E2 0, E3 0, E4 0}
LIN {X 590.525, Y 331.073, Z 390.319, A -106.87, B 85.042, C -82.235, E1 0, E2 0, E3 0, E4 0}
LIN {X 589.274, Y 327.373, Z 390.658, A -106.87, B 85.042, C -82.235, E1 0, E2 0, E3 0, E4 0}
LIN {X 589.277, Y 327.253, Z 390.668, A -106.87, B 85.042, C -82.235, E1 0, E2 0, E3 0, E4 0}
LIN {X 586.482, Y 321.496, Z 391.216, A -106.87, B 85.042, C -82.235, E1 0, E2 0, E3 0, E4 0}
LIN {X 585.884, Y 319.472, Z 391.399, A -106.87, B 85.042, C -82.235, E1 0, E2 0, E3 0, E4 0}
LIN {X 584.756, Y 317.738, Z 391.572, A -106.87, B 85.042, C -82.235, E1 0, E2 0, E3 0, E4 0}
LIN {X 560.637, Y 265.269, Z 396.535, A -106.87, B 85.042, C -82.235, E1 0, E2 0, E3 0, E4 0}
LIN {X 559.469, Y 262.754, Z 396.773, A -106.87, B 85.042, C -82.235, E1 0, E2 0, E3 0, E4 0}
LIN {X 557.985, Y 263.322, Z 396.763, A -106.87, B 85.042, C -82.235, E1 0, E2 0, E3 0, E4 0}
LIN {X 557.364, Y 263.333, Z 396.778, A -106.87, B 85.042, C -82.235, E1 0, E2 0, E3 0, E4 0}
LIN {X 556.928, Y 263.837, Z 396.747, A -106.87, B 85.042, C -82.235, E1 0, E2 0, E3 0, E4 0}
LIN {X 556.637, Y 265.071, Z 396.652, A -106.87, B 85.042, C -82.235, E1 0, E2 0, E3 0, E4 0}
LIN {X 558.536, Y 268.72, Z 396.302, A -106.87, B 85.042, C -82.235, E1 0, E2 0, E3 0, E4 0}
LIN {X 558.483, Y 272.448, Z 395.993, A -106.87, B 85.042, C -82.235, E1 0, E2 0, E3 0, E4 0}
LIN {X 558.774, Y 276.473, Z 395.652, A -106.87, B 85.042, C -82.235, E1 0, E2 0, E3 0, E4 0}
LIN {X 560.41, Y 309.31, Z 392.885, A -106.87, B 85.042, C -82.235, E1 0, E2 0, E3 0, E4 0}
LIN {X 560.056, Y 314.193, Z 392.488, A -106.87, B 85.042, C -82.235, E1 0, E2 0, E3 0, E4 0}
LIN {X 560.453, Y 315.79, Z 392.345, A -106.87, B 85.042, C -82.235, E1 0, E2 0, E3 0, E4 0}
LIN {X 560.371, Y 316.818, Z 392.262, A -106.87, B 85.042, C -82.235, E1 0, E2 0, E3 0, E4 0}
LIN {X 560.337, Y 316.887, Z 392.257, A -106.87, B 85.042, C -82.235, E1 0, E2 0, E3 0, E4 0}
LIN {X 560.705, Y 330.331, Z 391.132, A -106.87, B 85.042, C -82.235, E1 0, E2 0, E3 0, E4 0}
LIN {X 560.629, Y 330.491, Z 391.12, A -106.87, B 85.042, C -82.235, E1 0, E2 0, E3 0, E4 0}
LIN {X 559.682, Y 335.797, Z 390.704, A -106.87, B 85.042, C -82.235, E1 0, E2 0, E3 0, E4 0}
LIN {X 560.626, Y 348.934, Z 389.589, A -106.87, B 85.042, C -82.235, E1 0, E2 0, E3 0, E4 0}
LIN {X 561.407, Y 349.668, Z 389.509, A -106.87, B 85.042, C -82.235, E1 0, E2 0, E3 0, E4 0}
LIN {X 561.545, Y 349.624, Z 389.509, A -106.87, B 85.042, C -82.235, E1 0, E2 0, E3 0, E4 0}
LIN {X 562.104, Y 349.659, Z 389.492, A -106.87, B 85.042, C -82.235, E1 0, E2 0, E3 0, E4 0}
LIN {X 567.818, Y 348.066, Z 389.48, A -106.87, B 85.042, C -82.235, E1 0, E2 0, E3 0, E4 0}
LIN {X 571.64, Y 346.276, Z 389.533, A -106.87, B 85.042, C -82.235, E1 0, E2 0, E3 0, E4 0}
LIN {X 573.859, Y 345.883, Z 389.51, A -106.87, B 85.042, C -82.235, E1 0, E2 0, E3 0, E4 0}
LIN {X 574.016, Y 345.902, Z 389.504, A -106.87, B 85.042, C -82.235, E1 0, E2 0, E3 0, E4 0}
LIN {X 578.013, Y 344.835, Z 389.492, A -106.87, B 85.042, C -82.235, E1 0, E2 0, E3 0, E4 0}
LIN {X 578.154, Y 344.821, Z 389.49, A -106.87, B 85.042, C -82.235, E1 0, E2 0, E3 0, E4 0}
LIN {X 591.513, Y 334.971, Z 389.971, A -106.87, B 85.042, C -82.235, E1 0, E2 0, E3 0, E4 0}
LIN {X 591.458, Y 334.791, Z 387.805, A -106.87, B 85.042, C -82.235, E1 0, E2 0, E3 0, E4 0}
LIN {X 559.71, Y 349.33, Z 387.397, A -106.87, B 85.042, C -82.235, E1 0, E2 0, E3 0, E4 0}
LIN {X 559.592, Y 343.906, Z 387.851, A -106.87, B 85.042, C -82.235, E1 0, E2 0, E3 0, E4 0}
LIN {X 590.67, Y 329.673, Z 388.25, A -106.87, B 85.042, C -82.235, E1 0, E2 0, E3 0, E4 0}
LIN {X 590.375, Y 324.329, Z 388.701, A -106.87, B 85.042, C -82.235, E1 0, E2 0, E3 0, E4 0}
LIN {X 559.534, Y 338.453, Z 388.305, A -106.87, B 85.042, C -82.235, E1 0, E2 0, E3 0, E4 0}
LIN {X 560.275, Y 332.634, Z 388.769, A -106.87, B 85.042, C -82.235, E1 0, E2 0, E3 0, E4 0}
LIN {X 588.135, Y 319.875, Z 389.127, A -106.87, B 85.042, C -82.235, E1 0, E2 0, E3 0, E4 0}
LIN {X 586.099, Y 315.329, Z 389.556, A -106.87, B 85.042, C -82.235, E1 0, E2 0, E3 0, E4 0}
LIN {X 560.391, Y 327.102, Z 389.226, A -106.87, B 85.042, C -82.235, E1 0, E2 0, E3 0, E4 0}
LIN {X 560.214, Y 321.704, Z 389.678, A -106.87, B 85.042, C -82.235, E1 0, E2 0, E3 0, E4 0}
LIN {X 583.936, Y 310.84, Z 389.983, A -106.87, B 85.042, C -82.235, E1 0, E2 0, E3 0, E4 0}
LIN {X 582.291, Y 306.114, Z 390.417, A -106.87, B 85.042, C -82.235, E1 0, E2 0, E3 0, E4 0}
LIN {X 560.331, Y 316.171, Z 390.135, A -106.87, B 85.042, C -82.235, E1 0, E2 0, E3 0, E4 0}
LIN {X 560.297, Y 310.707, Z 390.589, A -106.87, B 85.042, C -82.235, E1 0, E2 0, E3 0, E4 0}
LIN {X 580.017, Y 301.677, Z 390.843, A -106.87, B 85.042, C -82.235, E1 0, E2 0, E3 0, E4 0}
LIN {X 578.013, Y 297.115, Z 391.272, A -106.87, B 85.042, C -82.235, E1 0, E2 0, E3 0, E4 0}
LIN {X 560.013, Y 305.358, Z 391.04, A -106.87, B 85.042, C -82.235, E1 0, E2 0, E3 0, E4 0}
LIN {X 559.762, Y 299.994, Z 391.492, A -106.87, B 85.042, C -82.235, E1 0, E2 0, E3 0, E4 0}
LIN {X 576.129, Y 292.499, Z 391.702, A -106.87, B 85.042, C -82.235, E1 0, E2 0, E3 0, E4 0}
LIN {X 574.036, Y 287.978, Z 392.13, A -106.87, B 85.042, C -82.235, E1 0, E2 0, E3 0, E4 0}
LIN {X 559.967, Y 294.421, Z 391.95, A -106.87, B 85.042, C -82.235, E1 0, E2 0, E3 0, E4 0}
LIN {X 559.555, Y 289.131, Z 392.399, A -106.87, B 85.042, C -82.235, E1 0, E2 0, E3 0, E4 0}
LIN {X 571.861, Y 283.495, Z 392.557, A -106.87, B 85.042, C -82.235, E1 0, E2 0, E3 0, E4 0}
LIN {X 570.155, Y 278.797, Z 392.99, A -106.87, B 85.042, C -82.235, E1 0, E2 0, E3 0, E4 0}
LIN {X 558.897, Y 283.953, Z 392.846, A -106.87, B 85.042, C -82.235, E1 0, E2 0, E3 0, E4 0}
LIN {X 558.735, Y 278.548, Z 393.298, A -106.87, B 85.042, C -82.235, E1 0, E2 0, E3 0, E4 0}
LIN {X 568.069, Y 274.273, Z 393.418, A -106.87, B 85.042, C -82.235, E1 0, E2 0, E3 0, E4 0}
LIN {X 565.547, Y 269.949, Z 393.841, A -106.87, B 85.042, C -82.235, E1 0, E2 0, E3 0, E4 0}
LIN {X 558.409, Y 273.218, Z 393.749, A -106.87, B 85.042, C -82.235, E1 0, E2 0, E3 0, E4 0}
LIN {X 558.269, Y 267.803, Z 394.202, A -106.87, B 85.042, C -82.235, E1 0, E2 0, E3 0, E4 0}
LIN {X 563.367, Y 265.468, Z 394.268, A -106.87, B 85.042, C -82.235, E1 0, E2 0, E3 0, E4 0}
LIN {X 578.054, Y 344.547, Z 387.333, A -106.87, B 85.042, C -82.235, E1 0, E2 0, E3 0, E4 0}
LIN {X 579.483, Y 343.857, Z 387.354, A -106.87, B 85.042, C -82.235, E1 0, E2 0, E3 0, E4 0}
LIN {X 582.999, Y 343.537, Z 387.292, A -106.87, B 85.042, C -82.235, E1 0, E2 0, E3 0, E4 0}
LIN {X 589.72, Y 339.527, Z 387.456, A -106.87, B 85.042, C -82.235, E1 0, E2 0, E3 0, E4 0}
LIN {X 592.084, Y 338.405, Z 387.489, A -106.87, B 85.042, C -82.235, E1 0, E2 0, E3 0, E4 0}
LIN {X 592.184, Y 338.328, Z 387.493, A -106.87, B 85.042, C -82.235, E1 0, E2 0, E3 0, E4 0}
LIN {X 592.479, Y 337.405, Z 387.563, A -106.87, B 85.042, C -82.235, E1 0, E2 0, E3 0, E4 0}
LIN {X 592.482, Y 336.289, Z 387.655, A -106.87, B 85.042, C -82.235, E1 0, E2 0, E3 0, E4 0}
LIN {X 592.012, Y 335.373, Z 387.743, A -106.87, B 85.042, C -82.235, E1 0, E2 0, E3 0, E4 0}
LIN {X 591.087, Y 334.318, Z 387.854, A -106.87, B 85.042, C -82.235, E1 0, E2 0, E3 0, E4 0}
LIN {X 590.52, Y 332.895, Z 387.986, A -106.87, B 85.042, C -82.235, E1 0, E2 0, E3 0, E4 0}
LIN {X 590.471, Y 331.717, Z 388.085, A -106.87, B 85.042, C -82.235, E1 0, E2 0, E3 0, E4 0}
LIN {X 590.457, Y 331.681, Z 388.089, A -106.87, B 85.042, C -82.235, E1 0, E2 0, E3 0, E4 0}
LIN {X 591.003, Y 326.86, Z 388.475, A -106.87, B 85.042, C -82.235, E1 0, E2 0, E3 0, E4 0}
LIN {X 591.011, Y 326.842, Z 388.477, A -106.87, B 85.042, C -82.235, E1 0, E2 0, E3 0, E4 0}
LIN {X 584.17, Y 311.316, Z 389.938, A -106.87, B 85.042, C -82.235, E1 0, E2 0, E3 0, E4 0}
LIN {X 562.207, Y 262.849, Z 394.514, A -106.87, B 85.042, C -82.235, E1 0, E2 0, E3 0, E4 0}
LIN {X 561.809, Y 262.793, Z 394.529, A -106.87, B 85.042, C -82.235, E1 0, E2 0, E3 0, E4 0}
LIN {X 561.776, Y 262.679, Z 394.539, A -106.87, B 85.042, C -82.235, E1 0, E2 0, E3 0, E4 0}
LIN {X 560.373, Y 262.384, Z 394.599, A -106.87, B 85.042, C -82.235, E1 0, E2 0, E3 0, E4 0}
LIN {X 557.931, Y 263.142, Z 394.598, A -106.87, B 85.042, C -82.235, E1 0, E2 0, E3 0, E4 0}
LIN {X 557.309, Y 263.153, Z 394.612, A -106.87, B 85.042, C -82.235, E1 0, E2 0, E3 0, E4 0}
LIN {X 556.873, Y 263.657, Z 394.582, A -106.87, B 85.042, C -82.235, E1 0, E2 0, E3 0, E4 0}
LIN {X 556.582, Y 264.892, Z 394.486, A -106.87, B 85.042, C -82.235, E1 0, E2 0, E3 0, E4 0}
LIN {X 558.482, Y 268.54, Z 394.136, A -106.87, B 85.042, C -82.235, E1 0, E2 0, E3 0, E4 0}
LIN {X 558.428, Y 272.268, Z 393.828, A -106.87, B 85.042, C -82.235, E1 0, E2 0, E3 0, E4 0}
LIN {X 558.719, Y 276.293, Z 393.486, A -106.87, B 85.042, C -82.235, E1 0, E2 0, E3 0, E4 0}
LIN {X 560.356, Y 309.13, Z 390.719, A -106.87, B 85.042, C -82.235, E1 0, E2 0, E3 0, E4 0}
LIN {X 560.001, Y 314.013, Z 390.322, A -106.87, B 85.042, C -82.235, E1 0, E2 0, E3 0, E4 0}
LIN {X 560.399, Y 315.61, Z 390.18, A -106.87, B 85.042, C -82.235, E1 0, E2 0, E3 0, E4 0}
LIN {X 560.316, Y 316.639, Z 390.096, A -106.87, B 85.042, C -82.235, E1 0, E2 0, E3 0, E4 0}
LIN {X 560.282, Y 316.707, Z 390.091, A -106.87, B 85.042, C -82.235, E1 0, E2 0, E3 0, E4 0}
LIN {X 560.65, Y 330.151, Z 388.966, A -106.87, B 85.042, C -82.235, E1 0, E2 0, E3 0, E4 0}
LIN {X 560.574, Y 330.311, Z 388.955, A -106.87, B 85.042, C -82.235, E1 0, E2 0, E3 0, E4 0}
LIN {X 559.628, Y 335.617, Z 388.538, A -106.87, B 85.042, C -82.235, E1 0, E2 0, E3 0, E4 0}
LIN {X 559.701, Y 350.328, Z 387.315, A -106.87, B 85.042, C -82.235, E1 0, E2 0, E3 0, E4 0}
LIN {X 559.747, Y 351.933, Z 387.181, A -106.87, B 85.042, C -82.235, E1 0, E2 0, E3 0, E4 0}
LIN {X 560.288, Y 351.827, Z 387.176, A -106.87, B 85.042, C -82.235, E1 0, E2 0, E3 0, E4 0}
LIN {X 560.806, Y 351.531, Z 387.187, A -106.87, B 85.042, C -82.235, E1 0, E2 0, E3 0, E4 0}
LIN {X 561.998, Y 350.426, Z 387.249, A -106.87, B 85.042, C -82.235, E1 0, E2 0, E3 0, E4 0}
LIN {X 562.026, Y 350.382, Z 387.252, A -106.87, B 85.042, C -82.235, E1 0, E2 0, E3 0, E4 0}
LIN {X 561.967, Y 350.349, Z 387.256, A -106.87, B 85.042, C -82.235, E1 0, E2 0, E3 0, E4 0}
LIN {X 563.121, Y 349.12, Z 387.329, A -106.87, B 85.042, C -82.235, E1 0, E2 0, E3 0, E4 0}
LIN {X 565.545, Y 348.543, Z 387.316, A -106.87, B 85.042, C -82.235, E1 0, E2 0, E3 0, E4 0}
LIN {X 566.179, Y 348.545, Z 387.3, A -106.87, B 85.042, C -82.235, E1 0, E2 0, E3 0, E4 0}
LIN {X 571.537, Y 346.965, Z 387.296, A -106.87, B 85.042, C -82.235, E1 0, E2 0, E3 0, E4 0}
LIN {X 573.387, Y 346.803, Z 387.263, A -106.87, B 85.042, C -82.235, E1 0, E2 0, E3 0, E4 0}
LIN {X 578.054, Y 344.547, Z 387.333, A -106.87, B 85.042, C -82.235, E1 0, E2 0, E3 0, E4 0}
LIN {X 592.653, Y 334.244, Z 387.821, A -106.87, B 85.042, C -82.235, E1 0, E2 0, E3 0, E4 0}
LIN {X 592.599, Y 334.064, Z 385.655, A -106.87, B 85.042, C -82.235, E1 0, E2 0, E3 0, E4 0}
LIN {X 559.656, Y 349.151, Z 385.232, A -106.87, B 85.042, C -82.235, E1 0, E2 0, E3 0, E4 0}
LIN {X 559.537, Y 343.726, Z 385.685, A -106.87, B 85.042, C -82.235, E1 0, E2 0, E3 0, E4 0}
LIN {X 590.595, Y 329.503, Z 386.084, A -106.87, B 85.042, C -82.235, E1 0, E2 0, E3 0, E4 0}
LIN {X 591.766, Y 323.487, Z 386.554, A -106.87, B 85.042, C -82.235, E1 0, E2 0, E3 0, E4 0}
LIN {X 559.479, Y 338.273, Z 386.139, A -106.87, B 85.042, C -82.235, E1 0, E2 0, E3 0, E4 0}
LIN {X 560.221, Y 332.454, Z 386.604, A -106.87, B 85.042, C -82.235, E1 0, E2 0, E3 0, E4 0}
LIN {X 589.975, Y 318.828, Z 386.986, A -106.87, B 85.042, C -82.235, E1 0, E2 0, E3 0, E4 0}
LIN {X 587.746, Y 314.37, Z 387.412, A -106.87, B 85.042, C -82.235, E1 0, E2 0, E3 0, E4 0}
LIN {X 560.336, Y 326.922, Z 387.06, A -106.87, B 85.042, C -82.235, E1 0, E2 0, E3 0, E4 0}
LIN {X 560.159, Y 321.524, Z 387.513, A -106.87, B 85.042, C -82.235, E1 0, E2 0, E3 0, E4 0}
LIN {X 585.875, Y 309.747, Z 387.843, A -106.87, B 85.042, C -82.235, E1 0, E2 0, E3 0, E4 0}
LIN {X 583.52, Y 305.347, Z 388.267, A -106.87, B 85.042, C -82.235, E1 0, E2 0, E3 0, E4 0}
LIN {X 560.276, Y 315.991, Z 387.969, A -106.87, B 85.042, C -82.235, E1 0, E2 0, E3 0, E4 0}
LIN {X 560.242, Y 310.528, Z 388.423, A -106.87, B 85.042, C -82.235, E1 0, E2 0, E3 0, E4 0}
LIN {X 581.413, Y 300.832, Z 388.695, A -106.87, B 85.042, C -82.235, E1 0, E2 0, E3 0, E4 0}
LIN {X 579.293, Y 296.324, Z 389.123, A -106.87, B 85.042, C -82.235, E1 0, E2 0, E3 0, E4 0}
LIN {X 559.959, Y 305.178, Z 388.875, A -106.87, B 85.042, C -82.235, E1 0, E2 0, E3 0, E4 0}
LIN {X 559.707, Y 299.814, Z 389.326, A -106.87, B 85.042, C -82.235, E1 0, E2 0, E3 0, E4 0}
LIN {X 577.379, Y 291.721, Z 389.553, A -106.87, B 85.042, C -82.235, E1 0, E2 0, E3 0, E4 0}
LIN {X 575.441, Y 287.13, Z 389.983, A -106.87, B 85.042, C -82.235, E1 0, E2 0, E3 0, E4 0}
LIN {X 559.912, Y 294.241, Z 389.784, A -106.87, B 85.042, C -82.235, E1 0, E2 0, E3 0, E4 0}
LIN {X 559.5, Y 288.951, Z 390.233, A -106.87, B 85.042, C -82.235, E1 0, E2 0, E3 0, E4 0}
LIN {X 573.266, Y 282.647, Z 390.41, A -106.87, B 85.042, C -82.235, E1 0, E2 0, E3 0, E4 0}
LIN {X 571.449, Y 278, Z 390.842, A -106.87, B 85.042, C -82.235, E1 0, E2 0, E3 0, E4 0}
LIN {X 558.842, Y 283.773, Z 390.68, A -106.87, B 85.042, C -82.235, E1 0, E2 0, E3 0, E4 0}
LIN {X 558.68, Y 278.368, Z 391.133, A -106.87, B 85.042, C -82.235, E1 0, E2 0, E3 0, E4 0}
LIN {X 569.596, Y 273.369, Z 391.273, A -106.87, B 85.042, C -82.235, E1 0, E2 0, E3 0, E4 0}
LIN {X 567.256, Y 268.961, Z 391.698, A -106.87, B 85.042, C -82.235, E1 0, E2 0, E3 0, E4 0}
LIN {X 558.354, Y 273.038, Z 391.583, A -106.87, B 85.042, C -82.235, E1 0, E2 0, E3 0, E4 0}
LIN {X 558.215, Y 267.623, Z 392.036, A -106.87, B 85.042, C -82.235, E1 0, E2 0, E3 0, E4 0}
LIN {X 565.227, Y 264.411, Z 392.126, A -106.87, B 85.042, C -82.235, E1 0, E2 0, E3 0, E4 0}
LIN {X 578.093, Y 344.685, Z 385.138, A -106.87, B 85.042, C -82.235, E1 0, E2 0, E3 0, E4 0}
LIN {X 581.765, Y 343.606, Z 385.135, A -106.87, B 85.042, C -82.235, E1 0, E2 0, E3 0, E4 0}
LIN {X 585.237, Y 342.629, Z 385.129, A -106.87, B 85.042, C -82.235, E1 0, E2 0, E3 0, E4 0}
LIN {X 590.697, Y 339.656, Z 385.239, A -106.87, B 85.042, C -82.235, E1 0, E2 0, E3 0, E4 0}
LIN {X 590.878, Y 339.599, Z 385.239, A -106.87, B 85.042, C -82.235, E1 0, E2 0, E3 0, E4 0}
LIN {X 591.639, Y 339.106, Z 385.261, A -106.87, B 85.042, C -82.235, E1 0, E2 0, E3 0, E4 0}
LIN {X 592.19, Y 339.14, Z 385.244, A -106.87, B 85.042, C -82.235, E1 0, E2 0, E3 0, E4 0}
LIN {X 592.829, Y 338.985, Z 385.241, A -106.87, B 85.042, C -82.235, E1 0, E2 0, E3 0, E4 0}
LIN {X 593.167, Y 339.177, Z 385.216, A -106.87, B 85.042, C -82.235, E1 0, E2 0, E3 0, E4 0}
LIN {X 593.94, Y 338.906, Z 385.219, A -106.87, B 85.042, C -82.235, E1 0, E2 0, E3 0, E4 0}
LIN {X 594.312, Y 338.133, Z 385.274, A -106.87, B 85.042, C -82.235, E1 0, E2 0, E3 0, E4 0}
LIN {X 594.279, Y 337.59, Z 385.32, A -106.87, B 85.042, C -82.235, E1 0, E2 0, E3 0, E4 0}
LIN {X 591.557, Y 331.429, Z 385.9, A -106.87, B 85.042, C -82.235, E1 0, E2 0, E3 0, E4 0}
LIN {X 590.771, Y 330.581, Z 385.99, A -106.87, B 85.042, C -82.235, E1 0, E2 0, E3 0, E4 0}
LIN {X 590.721, Y 330.473, Z 386, A -106.87, B 85.042, C -82.235, E1 0, E2 0, E3 0, E4 0}
LIN {X 590.427, Y 328.472, Z 386.174, A -106.87, B 85.042, C -82.235, E1 0, E2 0, E3 0, E4 0}
LIN {X 591.777, Y 322.742, Z 386.615, A -106.87, B 85.042, C -82.235, E1 0, E2 0, E3 0, E4 0}
LIN {X 591.324, Y 321.434, Z 386.735, A -106.87, B 85.042, C -82.235, E1 0, E2 0, E3 0, E4 0}
LIN {X 591.306, Y 321.271, Z 386.749, A -106.87, B 85.042, C -82.235, E1 0, E2 0, E3 0, E4 0}
LIN {X 587.673, Y 314.241, Z 387.425, A -106.87, B 85.042, C -82.235, E1 0, E2 0, E3 0, E4 0}
LIN {X 587.622, Y 314.013, Z 387.445, A -106.87, B 85.042, C -82.235, E1 0, E2 0, E3 0, E4 0}
LIN {X 564.105, Y 262.205, Z 392.338, A -106.87, B 85.042, C -82.235, E1 0, E2 0, E3 0, E4 0}
LIN {X 563.033, Y 262.456, Z 392.344, A -106.87, B 85.042, C -82.235, E1 0, E2 0, E3 0, E4 0}
LIN {X 562.995, Y 262.523, Z 392.339, A -106.87, B 85.042, C -82.235, E1 0, E2 0, E3 0, E4 0}
LIN {X 562.204, Y 262.676, Z 392.347, A -106.87, B 85.042, C -82.235, E1 0, E2 0, E3 0, E4 0}
LIN {X 561.755, Y 262.613, Z 392.363, A -106.87, B 85.042, C -82.235, E1 0, E2 0, E3 0, E4 0}
LIN {X 561.722, Y 262.5, Z 392.373, A -106.87, B 85.042, C -82.235, E1 0, E2 0, E3 0, E4 0}
LIN {X 560.318, Y 262.204, Z 392.433, A -106.87, B 85.042, C -82.235, E1 0, E2 0, E3 0, E4 0}
LIN {X 557.876, Y 262.962, Z 392.432, A -106.87, B 85.042, C -82.235, E1 0, E2 0, E3 0, E4 0}
LIN {X 557.255, Y 262.973, Z 392.447, A -106.87, B 85.042, C -82.235, E1 0, E2 0, E3 0, E4 0}
LIN {X 556.819, Y 263.477, Z 392.416, A -106.87, B 85.042, C -82.235, E1 0, E2 0, E3 0, E4 0}
LIN {X 556.528, Y 264.712, Z 392.321, A -106.87, B 85.042, C -82.235, E1 0, E2 0, E3 0, E4 0}
LIN {X 558.427, Y 268.36, Z 391.97, A -106.87, B 85.042, C -82.235, E1 0, E2 0, E3 0, E4 0}
LIN {X 558.374, Y 272.088, Z 391.662, A -106.87, B 85.042, C -82.235, E1 0, E2 0, E3 0, E4 0}
LIN {X 558.665, Y 276.113, Z 391.32, A -106.87, B 85.042, C -82.235, E1 0, E2 0, E3 0, E4 0}
LIN {X 560.301, Y 308.951, Z 388.553, A -106.87, B 85.042, C -82.235, E1 0, E2 0, E3 0, E4 0}
LIN {X 559.947, Y 313.833, Z 388.157, A -106.87, B 85.042, C -82.235, E1 0, E2 0, E3 0, E4 0}
LIN {X 560.344, Y 315.43, Z 388.014, A -106.87, B 85.042, C -82.235, E1 0, E2 0, E3 0, E4 0}
LIN {X 560.262, Y 316.459, Z 387.931, A -106.87, B 85.042, C -82.235, E1 0, E2 0, E3 0, E4 0}
LIN {X 560.228, Y 316.527, Z 387.926, A -106.87, B 85.042, C -82.235, E1 0, E2 0, E3 0, E4 0}
LIN {X 560.596, Y 329.971, Z 386.8, A -106.87, B 85.042, C -82.235, E1 0, E2 0, E3 0, E4 0}
LIN {X 560.52, Y 330.132, Z 386.789, A -106.87, B 85.042, C -82.235, E1 0, E2 0, E3 0, E4 0}
LIN {X 559.573, Y 335.437, Z 386.372, A -106.87, B 85.042, C -82.235, E1 0, E2 0, E3 0, E4 0}
LIN {X 559.646, Y 350.148, Z 385.149, A -106.87, B 85.042, C -82.235, E1 0, E2 0, E3 0, E4 0}
LIN {X 559.669, Y 350.973, Z 385.08, A -106.87, B 85.042, C -82.235, E1 0, E2 0, E3 0, E4 0}
LIN {X 562.696, Y 350.203, Z 385.068, A -106.87, B 85.042, C -82.235, E1 0, E2 0, E3 0, E4 0}
LIN {X 564.995, Y 348.798, Z 385.127, A -106.87, B 85.042, C -82.235, E1 0, E2 0, E3 0, E4 0}
LIN {X 571.951, Y 347.004, Z 385.1, A -106.87, B 85.042, C -82.235, E1 0, E2 0, E3 0, E4 0}
LIN {X 578.075, Y 344.69, Z 385.138, A -106.87, B 85.042, C -82.235, E1 0, E2 0, E3 0, E4 0}
LIN {X 578.093, Y 344.685, Z 385.138, A -106.87, B 85.042, C -82.235, E1 0, E2 0, E3 0, E4 0}
LIN {X 595.541, Y 338.196, Z 385.238, A -106.87, B 85.042, C -82.235, E1 0, E2 0, E3 0, E4 0}
LIN {X 595.487, Y 338.016, Z 383.072, A -106.87, B 85.042, C -82.235, E1 0, E2 0, E3 0, E4 0}
LIN {X 590.709, Y 340.204, Z 383.011, A -106.87, B 85.042, C -82.235, E1 0, E2 0, E3 0, E4 0}
LIN {X 589.476, Y 340.768, Z 382.995, A -106.87, B 85.042, C -82.235, E1 0, E2 0, E3 0, E4 0}
LIN {X 589.454, Y 340.779, Z 382.995, A -106.87, B 85.042, C -82.235, E1 0, E2 0, E3 0, E4 0}
LIN {X 587.33, Y 341.759, Z 382.967, A -106.87, B 85.042, C -82.235, E1 0, E2 0, E3 0, E4 0}
LIN {X 587.192, Y 341.804, Z 382.966, A -106.87, B 85.042, C -82.235, E1 0, E2 0, E3 0, E4 0}
LIN {X 593.613, Y 333.395, Z 383.503, A -106.87, B 85.042, C -82.235, E1 0, E2 0, E3 0, E4 0}
LIN {X 559.601, Y 348.971, Z 383.066, A -106.87, B 85.042, C -82.235, E1 0, E2 0, E3 0, E4 0}
LIN {X 559.483, Y 343.546, Z 383.519, A -106.87, B 85.042, C -82.235, E1 0, E2 0, E3 0, E4 0}
LIN {X 591.916, Y 328.693, Z 383.936, A -106.87, B 85.042, C -82.235, E1 0, E2 0, E3 0, E4 0}
LIN {X 590.71, Y 323.766, Z 384.375, A -106.87, B 85.042, C -82.235, E1 0, E2 0, E3 0, E4 0}
LIN {X 559.425, Y 338.093, Z 383.974, A -106.87, B 85.042, C -82.235, E1 0, E2 0, E3 0, E4 0}
LIN {X 560.166, Y 332.274, Z 384.438, A -106.87, B 85.042, C -82.235, E1 0, E2 0, E3 0, E4 0}
LIN {X 589.837, Y 318.686, Z 384.819, A -106.87, B 85.042, C -82.235, E1 0, E2 0, E3 0, E4 0}
LIN {X 587.581, Y 314.24, Z 385.245, A -106.87, B 85.042, C -82.235, E1 0, E2 0, E3 0, E4 0}
LIN {X 560.282, Y 326.742, Z 384.894, A -106.87, B 85.042, C -82.235, E1 0, E2 0, E3 0, E4 0}
LIN {X 560.105, Y 321.344, Z 385.347, A -106.87, B 85.042, C -82.235, E1 0, E2 0, E3 0, E4 0}
LIN {X 586.643, Y 309.191, Z 385.688, A -106.87, B 85.042, C -82.235, E1 0, E2 0, E3 0, E4 0}
LIN {X 584.292, Y 304.788, Z 386.112, A -106.87, B 85.042, C -82.235, E1 0, E2 0, E3 0, E4 0}
LIN {X 560.222, Y 315.811, Z 385.803, A -106.87, B 85.042, C -82.235, E1 0, E2 0, E3 0, E4 0}
LIN {X 560.188, Y 310.348, Z 386.258, A -106.87, B 85.042, C -82.235, E1 0, E2 0, E3 0, E4 0}
LIN {X 582.051, Y 300.335, Z 386.539, A -106.87, B 85.042, C -82.235, E1 0, E2 0, E3 0, E4 0}
LIN {X 580.626, Y 295.509, Z 386.975, A -106.87, B 85.042, C -82.235, E1 0, E2 0, E3 0, E4 0}
LIN {X 559.904, Y 304.999, Z 386.709, A -106.87, B 85.042, C -82.235, E1 0, E2 0, E3 0, E4 0}
LIN {X 559.653, Y 299.634, Z 387.161, A -106.87, B 85.042, C -82.235, E1 0, E2 0, E3 0, E4 0}
LIN {X 578.384, Y 291.056, Z 387.401, A -106.87, B 85.042, C -82.235, E1 0, E2 0, E3 0, E4 0}
LIN {X 576.518, Y 286.432, Z 387.832, A -106.87, B 85.042, C -82.235, E1 0, E2 0, E3 0, E4 0}
LIN {X 559.858, Y 294.061, Z 387.618, A -106.87, B 85.042, C -82.235, E1 0, E2 0, E3 0, E4 0}
LIN {X 559.446, Y 288.771, Z 388.068, A -106.87, B 85.042, C -82.235, E1 0, E2 0, E3 0, E4 0}
LIN {X 574.126, Y 282.048, Z 388.256, A -106.87, B 85.042, C -82.235, E1 0, E2 0, E3 0, E4 0}
LIN {X 572.033, Y 277.527, Z 388.684, A -106.87, B 85.042, C -82.235, E1 0, E2 0, E3 0, E4 0}
LIN {X 558.788, Y 283.593, Z 388.514, A -106.87, B 85.042, C -82.235, E1 0, E2 0, E3 0, E4 0}
LIN {X 558.626, Y 278.188, Z 388.967, A -106.87, B 85.042, C -82.235, E1 0, E2 0, E3 0, E4 0}
LIN {X 569.067, Y 273.406, Z 389.101, A -106.87, B 85.042, C -82.235, E1 0, E2 0, E3 0, E4 0}
LIN {X 568.313, Y 268.272, Z 389.546, A -106.87, B 85.042, C -82.235, E1 0, E2 0, E3 0, E4 0}
LIN {X 558.3, Y 272.858, Z 389.418, A -106.87, B 85.042, C -82.235, E1 0, E2 0, E3 0, E4 0}
LIN {X 558.16, Y 267.443, Z 389.871, A -106.87, B 85.042, C -82.235, E1 0, E2 0, E3 0, E4 0}
LIN {X 565.88, Y 263.908, Z 389.97, A -106.87, B 85.042, C -82.235, E1 0, E2 0, E3 0, E4 0}
LIN {X 578.074, Y 344.594, Z 382.964, A -106.87, B 85.042, C -82.235, E1 0, E2 0, E3 0, E4 0}
LIN {X 580.473, Y 343.626, Z 382.984, A -106.87, B 85.042, C -82.235, E1 0, E2 0, E3 0, E4 0}
LIN {X 582.277, Y 343.737, Z 382.93, A -106.87, B 85.042, C -82.235, E1 0, E2 0, E3 0, E4 0}
LIN {X 589.179, Y 341.015, Z 382.982, A -106.87, B 85.042, C -82.235, E1 0, E2 0, E3 0, E4 0}
LIN {X 590.345, Y 340.154, Z 383.024, A -106.87, B 85.042, C -82.235, E1 0, E2 0, E3 0, E4 0}
LIN {X 591.196, Y 340.272, Z 382.993, A -106.87, B 85.042, C -82.235, E1 0, E2 0, E3 0, E4 0}
LIN {X 592.969, Y 341.913, Z 382.812, A -106.87, B 85.042, C -82.235, E1 0, E2 0, E3 0, E4 0}
LIN {X 593.237, Y 341.934, Z 382.803, A -106.87, B 85.042, C -82.235, E1 0, E2 0, E3 0, E4 0}
LIN {X 593.882, Y 341.729, Z 382.804, A -106.87, B 85.042, C -82.235, E1 0, E2 0, E3 0, E4 0}
LIN {X 595.749, Y 339.143, Z 382.972, A -106.87, B 85.042, C -82.235, E1 0, E2 0, E3 0, E4 0}
LIN {X 595.729, Y 338.584, Z 383.019, A -106.87, B 85.042, C -82.235, E1 0, E2 0, E3 0, E4 0}
LIN {X 593.453, Y 332.493, Z 383.582, A -106.87, B 85.042, C -82.235, E1 0, E2 0, E3 0, E4 0}
LIN {X 591.07, Y 327.076, Z 384.091, A -106.87, B 85.042, C -82.235, E1 0, E2 0, E3 0, E4 0}
LIN {X 590.924, Y 326.048, Z 384.18, A -106.87, B 85.042, C -82.235, E1 0, E2 0, E3 0, E4 0}
LIN {X 590.955, Y 325.873, Z 384.194, A -106.87, B 85.042, C -82.235, E1 0, E2 0, E3 0, E4 0}
LIN {X 590.892, Y 325.391, Z 384.236, A -106.87, B 85.042, C -82.235, E1 0, E2 0, E3 0, E4 0}
LIN {X 590.967, Y 324.851, Z 384.279, A -106.87, B 85.042, C -82.235, E1 0, E2 0, E3 0, E4 0}
LIN {X 590.604, Y 323.516, Z 384.399, A -106.87, B 85.042, C -82.235, E1 0, E2 0, E3 0, E4 0}
LIN {X 590.93, Y 321.435, Z 384.563, A -106.87, B 85.042, C -82.235, E1 0, E2 0, E3 0, E4 0}
LIN {X 589.249, Y 317.169, Z 384.96, A -106.87, B 85.042, C -82.235, E1 0, E2 0, E3 0, E4 0}
LIN {X 588.52, Y 316.413, Z 385.041, A -106.87, B 85.042, C -82.235, E1 0, E2 0, E3 0, E4 0}
LIN {X 588.468, Y 316.402, Z 385.043, A -106.87, B 85.042, C -82.235, E1 0, E2 0, E3 0, E4 0}
LIN {X 588.488, Y 316.343, Z 385.048, A -106.87, B 85.042, C -82.235, E1 0, E2 0, E3 0, E4 0}
LIN {X 587.587, Y 314.332, Z 385.237, A -106.87, B 85.042, C -82.235, E1 0, E2 0, E3 0, E4 0}
LIN {X 586.857, Y 309.713, Z 385.639, A -106.87, B 85.042, C -82.235, E1 0, E2 0, E3 0, E4 0}
LIN {X 583.181, Y 302.207, Z 386.355, A -106.87, B 85.042, C -82.235, E1 0, E2 0, E3 0, E4 0}
LIN {X 582.924, Y 301.995, Z 386.379, A -106.87, B 85.042, C -82.235, E1 0, E2 0, E3 0, E4 0}
LIN {X 581.491, Y 299.018, Z 386.662, A -106.87, B 85.042, C -82.235, E1 0, E2 0, E3 0, E4 0}
LIN {X 581.408, Y 297.87, Z 386.759, A -106.87, B 85.042, C -82.235, E1 0, E2 0, E3 0, E4 0}
LIN {X 578.204, Y 290.187, Z 387.478, A -106.87, B 85.042, C -82.235, E1 0, E2 0, E3 0, E4 0}
LIN {X 573.595, Y 281.022, Z 388.355, A -106.87, B 85.042, C -82.235, E1 0, E2 0, E3 0, E4 0}
LIN {X 573.548, Y 280.603, Z 388.391, A -106.87, B 85.042, C -82.235, E1 0, E2 0, E3 0, E4 0}
LIN {X 572.643, Y 279.242, Z 388.527, A -106.87, B 85.042, C -82.235, E1 0, E2 0, E3 0, E4 0}
LIN {X 571.951, Y 277.227, Z 388.711, A -106.87, B 85.042, C -82.235, E1 0, E2 0, E3 0, E4 0}
LIN {X 569.072, Y 273.422, Z 389.1, A -106.87, B 85.042, C -82.235, E1 0, E2 0, E3 0, E4 0}
LIN {X 568.993, Y 273.137, Z 389.125, A -106.87, B 85.042, C -82.235, E1 0, E2 0, E3 0, E4 0}
LIN {X 569.139, Y 270.666, Z 389.327, A -106.87, B 85.042, C -82.235, E1 0, E2 0, E3 0, E4 0}
LIN {X 568.999, Y 269.633, Z 389.416, A -106.87, B 85.042, C -82.235, E1 0, E2 0, E3 0, E4 0}
LIN {X 566.141, Y 264.708, Z 389.897, A -106.87, B 85.042, C -82.235, E1 0, E2 0, E3 0, E4 0}
LIN {X 566.139, Y 264.607, Z 389.905, A -106.87, B 85.042, C -82.235, E1 0, E2 0, E3 0, E4 0}
LIN {X 565.638, Y 263.254, Z 390.03, A -106.87, B 85.042, C -82.235, E1 0, E2 0, E3 0, E4 0}
LIN {X 565.632, Y 262.219, Z 390.116, A -106.87, B 85.042, C -82.235, E1 0, E2 0, E3 0, E4 0}
LIN {X 565.421, Y 261.614, Z 390.172, A -106.87, B 85.042, C -82.235, E1 0, E2 0, E3 0, E4 0}
LIN {X 562.978, Y 262.276, Z 390.178, A -106.87, B 85.042, C -82.235, E1 0, E2 0, E3 0, E4 0}
LIN {X 562.941, Y 262.344, Z 390.174, A -106.87, B 85.042, C -82.235, E1 0, E2 0, E3 0, E4 0}
LIN {X 562.149, Y 262.497, Z 390.181, A -106.87, B 85.042, C -82.235, E1 0, E2 0, E3 0, E4 0}
LIN {X 561.7, Y 262.433, Z 390.198, A -106.87, B 85.042, C -82.235, E1 0, E2 0, E3 0, E4 0}
LIN {X 561.667, Y 262.32, Z 390.208, A -106.87, B 85.042, C -82.235, E1 0, E2 0, E3 0, E4 0}
LIN {X 560.264, Y 262.024, Z 390.268, A -106.87, B 85.042, C -82.235, E1 0, E2 0, E3 0, E4 0}
LIN {X 557.821, Y 262.782, Z 390.266, A -106.87, B 85.042, C -82.235, E1 0, E2 0, E3 0, E4 0}
LIN {X 557.2, Y 262.793, Z 390.281, A -106.87, B 85.042, C -82.235, E1 0, E2 0, E3 0, E4 0}
LIN {X 556.764, Y 263.297, Z 390.25, A -106.87, B 85.042, C -82.235, E1 0, E2 0, E3 0, E4 0}
LIN {X 556.473, Y 264.532, Z 390.155, A -106.87, B 85.042, C -82.235, E1 0, E2 0, E3 0, E4 0}
LIN {X 558.372, Y 268.18, Z 389.804, A -106.87, B 85.042, C -82.235, E1 0, E2 0, E3 0, E4 0}
LIN {X 558.319, Y 271.909, Z 389.496, A -106.87, B 85.042, C -82.235, E1 0, E2 0, E3 0, E4 0}
LIN {X 558.61, Y 275.934, Z 389.154, A -106.87, B 85.042, C -82.235, E1 0, E2 0, E3 0, E4 0}
LIN {X 560.247, Y 308.771, Z 386.387, A -106.87, B 85.042, C -82.235, E1 0, E2 0, E3 0, E4 0}
LIN {X 559.892, Y 313.654, Z 385.991, A -106.87, B 85.042, C -82.235, E1 0, E2 0, E3 0, E4 0}
LIN {X 560.29, Y 315.25, Z 385.848, A -106.87, B 85.042, C -82.235, E1 0, E2 0, E3 0, E4 0}
LIN {X 560.207, Y 316.279, Z 385.765, A -106.87, B 85.042, C -82.235, E1 0, E2 0, E3 0, E4 0}
LIN {X 560.173, Y 316.348, Z 385.76, A -106.87, B 85.042, C -82.235, E1 0, E2 0, E3 0, E4 0}
LIN {X 560.541, Y 329.792, Z 384.635, A -106.87, B 85.042, C -82.235, E1 0, E2 0, E3 0, E4 0}
LIN {X 560.465, Y 329.952, Z 384.623, A -106.87, B 85.042, C -82.235, E1 0, E2 0, E3 0, E4 0}
LIN {X 559.519, Y 335.257, Z 384.206, A -106.87, B 85.042, C -82.235, E1 0, E2 0, E3 0, E4 0}
LIN {X 559.59, Y 350.005, Z 382.98, A -106.87, B 85.042, C -82.235, E1 0, E2 0, E3 0, E4 0}
LIN {X 559.619, Y 350.949, Z 382.901, A -106.87, B 85.042, C -82.235, E1 0, E2 0, E3 0, E4 0}
LIN {X 563.879, Y 349.843, Z 382.886, A -106.87, B 85.042, C -82.235, E1 0, E2 0, E3 0, E4 0}
LIN {X 564.46, Y 349.425, Z 382.906, A -106.87, B 85.042, C -82.235, E1 0, E2 0, E3 0, E4 0}
LIN {X 573.339, Y 346.166, Z 382.953, A -106.87, B 85.042, C -82.235, E1 0, E2 0, E3 0, E4 0}
LIN {X 573.58, Y 346.189, Z 382.945, A -106.87, B 85.042, C -82.235, E1 0, E2 0, E3 0, E4 0}
LIN {X 574.583, Y 345.722, Z 382.958, A -106.87, B 85.042, C -82.235, E1 0, E2 0, E3 0, E4 0}
LIN {X 575.53, Y 345.62, Z 382.943, A -106.87, B 85.042, C -82.235, E1 0, E2 0, E3 0, E4 0}
LIN {X 578.074, Y 344.594, Z 382.964, A -106.87, B 85.042, C -82.235, E1 0, E2 0, E3 0, E4 0}
LIN {X 585.744, Y 342.477, Z 382.947, A -106.87, B 85.042, C -82.235, E1 0, E2 0, E3 0, E4 0}
LIN {X 585.69, Y 342.297, Z 380.781, A -106.87, B 85.042, C -82.235, E1 0, E2 0, E3 0, E4 0}
LIN {X 595.86, Y 337.64, Z 380.912, A -106.87, B 85.042, C -82.235, E1 0, E2 0, E3 0, E4 0}
LIN {X 594.121, Y 332.957, Z 381.344, A -106.87, B 85.042, C -82.235, E1 0, E2 0, E3 0, E4 0}
LIN {X 559.547, Y 348.791, Z 380.9, A -106.87, B 85.042, C -82.235, E1 0, E2 0, E3 0, E4 0}
LIN {X 559.428, Y 343.366, Z 381.354, A -106.87, B 85.042, C -82.235, E1 0, E2 0, E3 0, E4 0}
LIN {X 592.527, Y 328.208, Z 381.779, A -106.87, B 85.042, C -82.235, E1 0, E2 0, E3 0, E4 0}
LIN {X 590.597, Y 323.613, Z 382.209, A -106.87, B 85.042, C -82.235, E1 0, E2 0, E3 0, E4 0}
LIN {X 559.37, Y 337.913, Z 381.808, A -106.87, B 85.042, C -82.235, E1 0, E2 0, E3 0, E4 0}
LIN {X 560.112, Y 332.095, Z 382.272, A -106.87, B 85.042, C -82.235, E1 0, E2 0, E3 0, E4 0}
LIN {X 588.46, Y 319.112, Z 382.636, A -106.87, B 85.042, C -82.235, E1 0, E2 0, E3 0, E4 0}
LIN {X 586.303, Y 314.621, Z 383.063, A -106.87, B 85.042, C -82.235, E1 0, E2 0, E3 0, E4 0}
LIN {X 560.227, Y 326.563, Z 382.728, A -106.87, B 85.042, C -82.235, E1 0, E2 0, E3 0, E4 0}
LIN {X 560.05, Y 321.164, Z 383.181, A -106.87, B 85.042, C -82.235, E1 0, E2 0, E3 0, E4 0}
LIN {X 584.878, Y 309.794, Z 383.5, A -106.87, B 85.042, C -82.235, E1 0, E2 0, E3 0, E4 0}
LIN {X 581.723, Y 305.76, Z 383.914, A -106.87, B 85.042, C -82.235, E1 0, E2 0, E3 0, E4 0}
LIN {X 560.167, Y 315.632, Z 383.638, A -106.87, B 85.042, C -82.235, E1 0, E2 0, E3 0, E4 0}
LIN {X 560.133, Y 310.168, Z 384.092, A -106.87, B 85.042, C -82.235, E1 0, E2 0, E3 0, E4 0}
LIN {X 579.732, Y 301.193, Z 384.344, A -106.87, B 85.042, C -82.235, E1 0, E2 0, E3 0, E4 0}
LIN {X 579.547, Y 295.798, Z 384.796, A -106.87, B 85.042, C -82.235, E1 0, E2 0, E3 0, E4 0}
LIN {X 559.85, Y 304.819, Z 384.543, A -106.87, B 85.042, C -82.235, E1 0, E2 0, E3 0, E4 0}
LIN {X 559.598, Y 299.455, Z 384.995, A -106.87, B 85.042, C -82.235, E1 0, E2 0, E3 0, E4 0}
LIN {X 578.574, Y 290.764, Z 385.238, A -106.87, B 85.042, C -82.235, E1 0, E2 0, E3 0, E4 0}
LIN {X 576.586, Y 286.196, Z 385.668, A -106.87, B 85.042, C -82.235, E1 0, E2 0, E3 0, E4 0}
LIN {X 559.803, Y 293.882, Z 385.452, A -106.87, B 85.042, C -82.235, E1 0, E2 0, E3 0, E4 0}
LIN {X 559.391, Y 288.591, Z 385.902, A -106.87, B 85.042, C -82.235, E1 0, E2 0, E3 0, E4 0}
LIN {X 572.142, Y 282.752, Z 386.066, A -106.87, B 85.042, C -82.235, E1 0, E2 0, E3 0, E4 0}
LIN {X 569.938, Y 278.282, Z 386.492, A -106.87, B 85.042, C -82.235, E1 0, E2 0, E3 0, E4 0}
LIN {X 558.733, Y 283.413, Z 386.348, A -106.87, B 85.042, C -82.235, E1 0, E2 0, E3 0, E4 0}
LIN {X 558.571, Y 278.008, Z 386.801, A -106.87, B 85.042, C -82.235, E1 0, E2 0, E3 0, E4 0}
LIN {X 568.101, Y 273.644, Z 386.924, A -106.87, B 85.042, C -82.235, E1 0, E2 0, E3 0, E4 0}
LIN {X 566.212, Y 269.03, Z 387.354, A -106.87, B 85.042, C -82.235, E1 0, E2 0, E3 0, E4 0}
LIN {X 558.245, Y 272.678, Z 387.252, A -106.87, B 85.042, C -82.235, E1 0, E2 0, E3 0, E4 0}
LIN {X 558.106, Y 267.263, Z 387.705, A -106.87, B 85.042, C -82.235, E1 0, E2 0, E3 0, E4 0}
LIN {X 564.188, Y 264.478, Z 387.783, A -106.87, B 85.042, C -82.235, E1 0, E2 0, E3 0, E4 0}
LIN {X 578.225, Y 345.062, Z 380.74, A -106.87, B 85.042, C -82.235, E1 0, E2 0, E3 0, E4 0}
LIN {X 580.668, Y 344.289, Z 380.742, A -106.87, B 85.042, C -82.235, E1 0, E2 0, E3 0, E4 0}
LIN {X 580.757, Y 344.214, Z 380.746, A -106.87, B 85.042, C -82.235, E1 0, E2 0, E3 0, E4 0}
LIN {X 589.523, Y 341.622, Z 380.741, A -106.87, B 85.042, C -82.235, E1 0, E2 0, E3 0, E4 0}
LIN {X 592.788, Y 342.866, Z 380.555, A -106.87, B 85.042, C -82.235, E1 0, E2 0, E3 0, E4 0}
LIN {X 593.789, Y 342.774, Z 380.538, A -106.87, B 85.042, C -82.235, E1 0, E2 0, E3 0, E4 0}
LIN {X 596.333, Y 339.427, Z 380.751, A -106.87, B 85.042, C -82.235, E1 0, E2 0, E3 0, E4 0}
LIN {X 596.393, Y 338.602, Z 380.818, A -106.87, B 85.042, C -82.235, E1 0, E2 0, E3 0, E4 0}
LIN {X 596.15, Y 338.291, Z 380.85, A -106.87, B 85.042, C -82.235, E1 0, E2 0, E3 0, E4 0}
LIN {X 589.935, Y 321.757, Z 382.379, A -106.87, B 85.042, C -82.235, E1 0, E2 0, E3 0, E4 0}
LIN {X 588.451, Y 320.682, Z 382.506, A -106.87, B 85.042, C -82.235, E1 0, E2 0, E3 0, E4 0}
LIN {X 588.339, Y 320.583, Z 382.517, A -106.87, B 85.042, C -82.235, E1 0, E2 0, E3 0, E4 0}
LIN {X 588.495, Y 319.2, Z 382.628, A -106.87, B 85.042, C -82.235, E1 0, E2 0, E3 0, E4 0}
LIN {X 588.102, Y 317.807, Z 382.754, A -106.87, B 85.042, C -82.235, E1 0, E2 0, E3 0, E4 0}
LIN {X 586.375, Y 314.907, Z 383.038, A -106.87, B 85.042, C -82.235, E1 0, E2 0, E3 0, E4 0}
LIN {X 585.044, Y 311.19, Z 383.38, A -106.87, B 85.042, C -82.235, E1 0, E2 0, E3 0, E4 0}
LIN {X 584.835, Y 310.357, Z 383.454, A -106.87, B 85.042, C -82.235, E1 0, E2 0, E3 0, E4 0}
LIN {X 585.036, Y 307.713, Z 383.669, A -106.87, B 85.042, C -82.235, E1 0, E2 0, E3 0, E4 0}
LIN {X 584.476, Y 306.637, Z 383.772, A -106.87, B 85.042, C -82.235, E1 0, E2 0, E3 0, E4 0}
LIN {X 583.255, Y 305.603, Z 383.889, A -106.87, B 85.042, C -82.235, E1 0, E2 0, E3 0, E4 0}
LIN {X 581.738, Y 305.813, Z 383.91, A -106.87, B 85.042, C -82.235, E1 0, E2 0, E3 0, E4 0}
LIN {X 581.353, Y 304.925, Z 383.993, A -106.87, B 85.042, C -82.235, E1 0, E2 0, E3 0, E4 0}
LIN {X 581.369, Y 304.825, Z 384.001, A -106.87, B 85.042, C -82.235, E1 0, E2 0, E3 0, E4 0}
LIN {X 578.811, Y 299.406, Z 384.515, A -106.87, B 85.042, C -82.235, E1 0, E2 0, E3 0, E4 0}
LIN {X 578.907, Y 298.68, Z 384.573, A -106.87, B 85.042, C -82.235, E1 0, E2 0, E3 0, E4 0}
LIN {X 578.288, Y 298.142, Z 384.633, A -106.87, B 85.042, C -82.235, E1 0, E2 0, E3 0, E4 0}
LIN {X 578.249, Y 297.915, Z 384.653, A -106.87, B 85.042, C -82.235, E1 0, E2 0, E3 0, E4 0}
LIN {X 579.723, Y 295.37, Z 384.827, A -106.87, B 85.042, C -82.235, E1 0, E2 0, E3 0, E4 0}
LIN {X 579.755, Y 293.716, Z 384.964, A -106.87, B 85.042, C -82.235, E1 0, E2 0, E3 0, E4 0}
LIN {X 577.603, Y 288.677, Z 385.436, A -106.87, B 85.042, C -82.235, E1 0, E2 0, E3 0, E4 0}
LIN {X 577.571, Y 287.757, Z 385.513, A -106.87, B 85.042, C -82.235, E1 0, E2 0, E3 0, E4 0}
LIN {X 577.221, Y 286.752, Z 385.606, A -106.87, B 85.042, C -82.235, E1 0, E2 0, E3 0, E4 0}
LIN {X 574.195, Y 284.525, Z 385.867, A -106.87, B 85.042, C -82.235, E1 0, E2 0, E3 0, E4 0}
LIN {X 572.668, Y 284.311, Z 385.923, A -106.87, B 85.042, C -82.235, E1 0, E2 0, E3 0, E4 0}
LIN {X 572.649, Y 284.286, Z 385.925, A -106.87, B 85.042, C -82.235, E1 0, E2 0, E3 0, E4 0}
LIN {X 572.63, Y 284.211, Z 385.932, A -106.87, B 85.042, C -82.235, E1 0, E2 0, E3 0, E4 0}
LIN {X 572.761, Y 283.503, Z 385.988, A -106.87, B 85.042, C -82.235, E1 0, E2 0, E3 0, E4 0}
LIN {X 572.473, Y 283.095, Z 386.029, A -106.87, B 85.042, C -82.235, E1 0, E2 0, E3 0, E4 0}
LIN {X 572.453, Y 282.918, Z 386.044, A -106.87, B 85.042, C -82.235, E1 0, E2 0, E3 0, E4 0}
LIN {X 571.729, Y 282.51, Z 386.096, A -106.87, B 85.042, C -82.235, E1 0, E2 0, E3 0, E4 0}
LIN {X 571.128, Y 280.479, Z 386.28, A -106.87, B 85.042, C -82.235, E1 0, E2 0, E3 0, E4 0}
LIN {X 570.501, Y 279.939, Z 386.341, A -106.87, B 85.042, C -82.235, E1 0, E2 0, E3 0, E4 0}
LIN {X 569.996, Y 278.819, Z 386.446, A -106.87, B 85.042, C -82.235, E1 0, E2 0, E3 0, E4 0}
LIN {X 569.775, Y 277.307, Z 386.577, A -106.87, B 85.042, C -82.235, E1 0, E2 0, E3 0, E4 0}
LIN {X 569.765, Y 276.853, Z 386.615, A -106.87, B 85.042, C -82.235, E1 0, E2 0, E3 0, E4 0}
LIN {X 569.675, Y 276.73, Z 386.628, A -106.87, B 85.042, C -82.235, E1 0, E2 0, E3 0, E4 0}
LIN {X 569.319, Y 276.46, Z 386.659, A -106.87, B 85.042, C -82.235, E1 0, E2 0, E3 0, E4 0}
LIN {X 568.363, Y 273.999, Z 386.887, A -106.87, B 85.042, C -82.235, E1 0, E2 0, E3 0, E4 0}
LIN {X 567.421, Y 273.015, Z 386.993, A -106.87, B 85.042, C -82.235, E1 0, E2 0, E3 0, E4 0}
LIN {X 566.259, Y 269.076, Z 387.349, A -106.87, B 85.042, C -82.235, E1 0, E2 0, E3 0, E4 0}
LIN {X 565.823, Y 268.646, Z 387.396, A -106.87, B 85.042, C -82.235, E1 0, E2 0, E3 0, E4 0}
LIN {X 565.031, Y 266.854, Z 387.564, A -106.87, B 85.042, C -82.235, E1 0, E2 0, E3 0, E4 0}
LIN {X 564.945, Y 266.782, Z 387.573, A -106.87, B 85.042, C -82.235, E1 0, E2 0, E3 0, E4 0}
LIN {X 564.782, Y 266.31, Z 387.616, A -106.87, B 85.042, C -82.235, E1 0, E2 0, E3 0, E4 0}
LIN {X 564.64, Y 266.046, Z 387.641, A -106.87, B 85.042, C -82.235, E1 0, E2 0, E3 0, E4 0}
LIN {X 564.48, Y 265.148, Z 387.72, A -106.87, B 85.042, C -82.235, E1 0, E2 0, E3 0, E4 0}
LIN {X 564.317, Y 264.983, Z 387.738, A -106.87, B 85.042, C -82.235, E1 0, E2 0, E3 0, E4 0}
LIN {X 564.148, Y 264.319, Z 387.797, A -106.87, B 85.042, C -82.235, E1 0, E2 0, E3 0, E4 0}
LIN {X 563.833, Y 264.032, Z 387.829, A -106.87, B 85.042, C -82.235, E1 0, E2 0, E3 0, E4 0}
LIN {X 563.558, Y 262.047, Z 388.001, A -106.87, B 85.042, C -82.235, E1 0, E2 0, E3 0, E4 0}
LIN {X 563.593, Y 261.947, Z 388.008, A -106.87, B 85.042, C -82.235, E1 0, E2 0, E3 0, E4 0}
LIN {X 562.924, Y 262.096, Z 388.013, A -106.87, B 85.042, C -82.235, E1 0, E2 0, E3 0, E4 0}
LIN {X 562.886, Y 262.164, Z 388.008, A -106.87, B 85.042, C -82.235, E1 0, E2 0, E3 0, E4 0}
LIN {X 562.095, Y 262.317, Z 388.015, A -106.87, B 85.042, C -82.235, E1 0, E2 0, E3 0, E4 0}
LIN {X 561.646, Y 262.253, Z 388.032, A -106.87, B 85.042, C -82.235, E1 0, E2 0, E3 0, E4 0}
LIN {X 561.613, Y 262.14, Z 388.042, A -106.87, B 85.042, C -82.235, E1 0, E2 0, E3 0, E4 0}
LIN {X 560.209, Y 261.844, Z 388.102, A -106.87, B 85.042, C -82.235, E1 0, E2 0, E3 0, E4 0}
LIN {X 557.767, Y 262.603, Z 388.1, A -106.87, B 85.042, C -82.235, E1 0, E2 0, E3 0, E4 0}
LIN {X 557.146, Y 262.614, Z 388.115, A -106.87, B 85.042, C -82.235, E1 0, E2 0, E3 0, E4 0}
LIN {X 556.71, Y 263.117, Z 388.084, A -106.87, B 85.042, C -82.235, E1 0, E2 0, E3 0, E4 0}
LIN {X 556.419, Y 264.352, Z 387.989, A -106.87, B 85.042, C -82.235, E1 0, E2 0, E3 0, E4 0}
LIN {X 558.318, Y 268.001, Z 387.638, A -106.87, B 85.042, C -82.235, E1 0, E2 0, E3 0, E4 0}
LIN {X 558.265, Y 271.729, Z 387.33, A -106.87, B 85.042, C -82.235, E1 0, E2 0, E3 0, E4 0}
LIN {X 558.556, Y 275.754, Z 386.989, A -106.87, B 85.042, C -82.235, E1 0, E2 0, E3 0, E4 0}
LIN {X 560.192, Y 308.591, Z 384.221, A -106.87, B 85.042, C -82.235, E1 0, E2 0, E3 0, E4 0}
LIN {X 559.838, Y 313.474, Z 383.825, A -106.87, B 85.042, C -82.235, E1 0, E2 0, E3 0, E4 0}
LIN {X 560.235, Y 315.07, Z 383.682, A -106.87, B 85.042, C -82.235, E1 0, E2 0, E3 0, E4 0}
LIN {X 560.153, Y 316.099, Z 383.599, A -106.87, B 85.042, C -82.235, E1 0, E2 0, E3 0, E4 0}
LIN {X 560.119, Y 316.168, Z 383.594, A -106.87, B 85.042, C -82.235, E1 0, E2 0, E3 0, E4 0}
LIN {X 560.487, Y 329.612, Z 382.469, A -106.87, B 85.042, C -82.235, E1 0, E2 0, E3 0, E4 0}
LIN {X 560.41, Y 329.772, Z 382.457, A -106.87, B 85.042, C -82.235, E1 0, E2 0, E3 0, E4 0}
LIN {X 559.464, Y 335.077, Z 382.041, A -106.87, B 85.042, C -82.235, E1 0, E2 0, E3 0, E4 0}
LIN {X 559.537, Y 349.789, Z 380.818, A -106.87, B 85.042, C -82.235, E1 0, E2 0, E3 0, E4 0}
LIN {X 559.581, Y 351.299, Z 380.691, A -106.87, B 85.042, C -82.235, E1 0, E2 0, E3 0, E4 0}
LIN {X 568.554, Y 348.927, Z 380.662, A -106.87, B 85.042, C -82.235, E1 0, E2 0, E3 0, E4 0}
LIN {X 574.563, Y 346.222, Z 380.735, A -106.87, B 85.042, C -82.235, E1 0, E2 0, E3 0, E4 0}
LIN {X 578.225, Y 345.062, Z 380.74, A -106.87, B 85.042, C -82.235, E1 0, E2 0, E3 0, E4 0}
LIN {X 593.159, Y 344.356, Z 380.422, A -106.87, B 85.042, C -82.235, E1 0, E2 0, E3 0, E4 0}
LIN {X 593.104, Y 344.177, Z 378.256, A -106.87, B 85.042, C -82.235, E1 0, E2 0, E3 0, E4 0}
LIN {X 594.492, Y 343.541, Z 378.274, A -106.87, B 85.042, C -82.235, E1 0, E2 0, E3 0, E4 0}
LIN {X 596.544, Y 337.122, Z 378.755, A -106.87, B 85.042, C -82.235, E1 0, E2 0, E3 0, E4 0}
LIN {X 582.784, Y 343.423, Z 378.579, A -106.87, B 85.042, C -82.235, E1 0, E2 0, E3 0, E4 0}
LIN {X 580.937, Y 344.27, Z 378.555, A -106.87, B 85.042, C -82.235, E1 0, E2 0, E3 0, E4 0}
LIN {X 581.065, Y 344.211, Z 378.557, A -106.87, B 85.042, C -82.235, E1 0, E2 0, E3 0, E4 0}
LIN {X 580.475, Y 344.481, Z 378.549, A -106.87, B 85.042, C -82.235, E1 0, E2 0, E3 0, E4 0}
LIN {X 579.041, Y 345.138, Z 378.531, A -106.87, B 85.042, C -82.235, E1 0, E2 0, E3 0, E4 0}
LIN {X 559.492, Y 348.611, Z 378.734, A -106.87, B 85.042, C -82.235, E1 0, E2 0, E3 0, E4 0}
LIN {X 594.56, Y 332.551, Z 379.185, A -106.87, B 85.042, C -82.235, E1 0, E2 0, E3 0, E4 0}
LIN {X 592.698, Y 327.925, Z 379.616, A -106.87, B 85.042, C -82.235, E1 0, E2 0, E3 0, E4 0}
LIN {X 559.374, Y 343.186, Z 379.188, A -106.87, B 85.042, C -82.235, E1 0, E2 0, E3 0, E4 0}
LIN {X 559.316, Y 337.734, Z 379.642, A -106.87, B 85.042, C -82.235, E1 0, E2 0, E3 0, E4 0}
LIN {X 590.885, Y 323.276, Z 380.047, A -106.87, B 85.042, C -82.235, E1 0, E2 0, E3 0, E4 0}
LIN {X 588.453, Y 318.911, Z 380.471, A -106.87, B 85.042, C -82.235, E1 0, E2 0, E3 0, E4 0}
LIN {X 560.057, Y 331.915, Z 380.106, A -106.87, B 85.042, C -82.235, E1 0, E2 0, E3 0, E4 0}
LIN {X 560.172, Y 326.383, Z 380.563, A -106.87, B 85.042, C -82.235, E1 0, E2 0, E3 0, E4 0}
LIN {X 586.315, Y 314.41, Z 380.898, A -106.87, B 85.042, C -82.235, E1 0, E2 0, E3 0, E4 0}
LIN {X 584.539, Y 309.745, Z 381.331, A -106.87, B 85.042, C -82.235, E1 0, E2 0, E3 0, E4 0}
LIN {X 559.996, Y 320.985, Z 381.015, A -106.87, B 85.042, C -82.235, E1 0, E2 0, E3 0, E4 0}
LIN {X 560.113, Y 315.452, Z 381.472, A -106.87, B 85.042, C -82.235, E1 0, E2 0, E3 0, E4 0}
LIN {X 581.922, Y 305.464, Z 381.752, A -106.87, B 85.042, C -82.235, E1 0, E2 0, E3 0, E4 0}
LIN {X 580.198, Y 300.774, Z 382.185, A -106.87, B 85.042, C -82.235, E1 0, E2 0, E3 0, E4 0}
LIN {X 560.079, Y 309.988, Z 381.926, A -106.87, B 85.042, C -82.235, E1 0, E2 0, E3 0, E4 0}
LIN {X 559.795, Y 304.639, Z 382.377, A -106.87, B 85.042, C -82.235, E1 0, E2 0, E3 0, E4 0}
LIN {X 578.145, Y 296.235, Z 382.613, A -106.87, B 85.042, C -82.235, E1 0, E2 0, E3 0, E4 0}
LIN {X 576.681, Y 291.427, Z 383.049, A -106.87, B 85.042, C -82.235, E1 0, E2 0, E3 0, E4 0}
LIN {X 559.544, Y 299.275, Z 382.829, A -106.87, B 85.042, C -82.235, E1 0, E2 0, E3 0, E4 0}
LIN {X 559.749, Y 293.702, Z 383.287, A -106.87, B 85.042, C -82.235, E1 0, E2 0, E3 0, E4 0}
LIN {X 574.511, Y 286.941, Z 383.476, A -106.87, B 85.042, C -82.235, E1 0, E2 0, E3 0, E4 0}
LIN {X 572.634, Y 282.322, Z 383.907, A -106.87, B 85.042, C -82.235, E1 0, E2 0, E3 0, E4 0}
LIN {X 559.337, Y 288.411, Z 383.736, A -106.87, B 85.042, C -82.235, E1 0, E2 0, E3 0, E4 0}
LIN {X 558.678, Y 283.234, Z 384.183, A -106.87, B 85.042, C -82.235, E1 0, E2 0, E3 0, E4 0}
LIN {X 570.65, Y 277.751, Z 384.336, A -106.87, B 85.042, C -82.235, E1 0, E2 0, E3 0, E4 0}
LIN {X 568.659, Y 273.184, Z 384.765, A -106.87, B 85.042, C -82.235, E1 0, E2 0, E3 0, E4 0}
LIN {X 558.517, Y 277.829, Z 384.635, A -106.87, B 85.042, C -82.235, E1 0, E2 0, E3 0, E4 0}
LIN {X 558.191, Y 272.499, Z 385.086, A -106.87, B 85.042, C -82.235, E1 0, E2 0, E3 0, E4 0}
LIN {X 566.713, Y 268.596, Z 385.196, A -106.87, B 85.042, C -82.235, E1 0, E2 0, E3 0, E4 0}
LIN {X 564.846, Y 263.972, Z 385.626, A -106.87, B 85.042, C -82.235, E1 0, E2 0, E3 0, E4 0}
LIN {X 558.051, Y 267.083, Z 385.539, A -106.87, B 85.042, C -82.235, E1 0, E2 0, E3 0, E4 0}
LIN {X 578.308, Y 345.308, Z 378.535, A -106.87, B 85.042, C -82.235, E1 0, E2 0, E3 0, E4 0}
LIN {X 588.99, Y 341.849, Z 378.553, A -106.87, B 85.042, C -82.235, E1 0, E2 0, E3 0, E4 0}
LIN {X 589.954, Y 342.094, Z 378.508, A -106.87, B 85.042, C -82.235, E1 0, E2 0, E3 0, E4 0}
LIN {X 593.725, Y 344.548, Z 378.21, A -106.87, B 85.042, C -82.235, E1 0, E2 0, E3 0, E4 0}
LIN {X 593.888, Y 344.542, Z 378.206, A -106.87, B 85.042, C -82.235, E1 0, E2 0, E3 0, E4 0}
LIN {X 594.007, Y 344.432, Z 378.212, A -106.87, B 85.042, C -82.235, E1 0, E2 0, E3 0, E4 0}
LIN {X 596.789, Y 339.493, Z 378.552, A -106.87, B 85.042, C -82.235, E1 0, E2 0, E3 0, E4 0}
LIN {X 597.141, Y 338.821, Z 378.599, A -106.87, B 85.042, C -82.235, E1 0, E2 0, E3 0, E4 0}
LIN {X 590.634, Y 322.329, Z 380.132, A -106.87, B 85.042, C -82.235, E1 0, E2 0, E3 0, E4 0}
LIN {X 590.308, Y 321.876, Z 380.178, A -106.87, B 85.042, C -82.235, E1 0, E2 0, E3 0, E4 0}
LIN {X 590.103, Y 321.752, Z 380.194, A -106.87, B 85.042, C -82.235, E1 0, E2 0, E3 0, E4 0}
LIN {X 589.39, Y 321.625, Z 380.222, A -106.87, B 85.042, C -82.235, E1 0, E2 0, E3 0, E4 0}
LIN {X 588.878, Y 321.185, Z 380.271, A -106.87, B 85.042, C -82.235, E1 0, E2 0, E3 0, E4 0}
LIN {X 588.431, Y 318.657, Z 380.493, A -106.87, B 85.042, C -82.235, E1 0, E2 0, E3 0, E4 0}
LIN {X 586.525, Y 314.981, Z 380.846, A -106.87, B 85.042, C -82.235, E1 0, E2 0, E3 0, E4 0}
LIN {X 583.84, Y 307.764, Z 381.513, A -106.87, B 85.042, C -82.235, E1 0, E2 0, E3 0, E4 0}
LIN {X 582.516, Y 306.031, Z 381.69, A -106.87, B 85.042, C -82.235, E1 0, E2 0, E3 0, E4 0}
LIN {X 582.109, Y 305.813, Z 381.718, A -106.87, B 85.042, C -82.235, E1 0, E2 0, E3 0, E4 0}
LIN {X 580.933, Y 303.898, Z 381.907, A -106.87, B 85.042, C -82.235, E1 0, E2 0, E3 0, E4 0}
LIN {X 580.029, Y 300.034, Z 382.25, A -106.87, B 85.042, C -82.235, E1 0, E2 0, E3 0, E4 0}
LIN {X 578.35, Y 296.958, Z 382.548, A -106.87, B 85.042, C -82.235, E1 0, E2 0, E3 0, E4 0}
LIN {X 577.765, Y 295.016, Z 382.724, A -106.87, B 85.042, C -82.235, E1 0, E2 0, E3 0, E4 0}
LIN {X 577.648, Y 294.819, Z 382.743, A -106.87, B 85.042, C -82.235, E1 0, E2 0, E3 0, E4 0}
LIN {X 576.904, Y 291.613, Z 383.028, A -106.87, B 85.042, C -82.235, E1 0, E2 0, E3 0, E4 0}
LIN {X 576.631, Y 291.386, Z 383.054, A -106.87, B 85.042, C -82.235, E1 0, E2 0, E3 0, E4 0}
LIN {X 575.619, Y 289.506, Z 383.235, A -106.87, B 85.042, C -82.235, E1 0, E2 0, E3 0, E4 0}
LIN {X 575.521, Y 289.46, Z 383.242, A -106.87, B 85.042, C -82.235, E1 0, E2 0, E3 0, E4 0}
LIN {X 575.022, Y 288.057, Z 383.371, A -106.87, B 85.042, C -82.235, E1 0, E2 0, E3 0, E4 0}
LIN {X 574.835, Y 287.859, Z 383.392, A -106.87, B 85.042, C -82.235, E1 0, E2 0, E3 0, E4 0}
LIN {X 574.437, Y 286.254, Z 383.535, A -106.87, B 85.042, C -82.235, E1 0, E2 0, E3 0, E4 0}
LIN {X 574.13, Y 285.862, Z 383.575, A -106.87, B 85.042, C -82.235, E1 0, E2 0, E3 0, E4 0}
LIN {X 574.043, Y 285.586, Z 383.6, A -106.87, B 85.042, C -82.235, E1 0, E2 0, E3 0, E4 0}
LIN {X 573.443, Y 285.117, Z 383.654, A -106.87, B 85.042, C -82.235, E1 0, E2 0, E3 0, E4 0}
LIN {X 573.096, Y 283.439, Z 383.802, A -106.87, B 85.042, C -82.235, E1 0, E2 0, E3 0, E4 0}
LIN {X 571.955, Y 280.538, Z 384.072, A -106.87, B 85.042, C -82.235, E1 0, E2 0, E3 0, E4 0}
LIN {X 571.695, Y 279.483, Z 384.166, A -106.87, B 85.042, C -82.235, E1 0, E2 0, E3 0, E4 0}
LIN {X 571.58, Y 279.352, Z 384.18, A -106.87, B 85.042, C -82.235, E1 0, E2 0, E3 0, E4 0}
LIN {X 563.992, Y 261.65, Z 385.841, A -106.87, B 85.042, C -82.235, E1 0, E2 0, E3 0, E4 0}
LIN {X 562.869, Y 261.917, Z 385.847, A -106.87, B 85.042, C -82.235, E1 0, E2 0, E3 0, E4 0}
LIN {X 562.832, Y 261.984, Z 385.842, A -106.87, B 85.042, C -82.235, E1 0, E2 0, E3 0, E4 0}
LIN {X 562.04, Y 262.137, Z 385.849, A -106.87, B 85.042, C -82.235, E1 0, E2 0, E3 0, E4 0}
LIN {X 561.591, Y 262.073, Z 385.866, A -106.87, B 85.042, C -82.235, E1 0, E2 0, E3 0, E4 0}
LIN {X 561.558, Y 261.96, Z 385.876, A -106.87, B 85.042, C -82.235, E1 0, E2 0, E3 0, E4 0}
LIN {X 560.155, Y 261.665, Z 385.936, A -106.87, B 85.042, C -82.235, E1 0, E2 0, E3 0, E4 0}
LIN {X 557.712, Y 262.423, Z 385.935, A -106.87, B 85.042, C -82.235, E1 0, E2 0, E3 0, E4 0}
LIN {X 557.091, Y 262.434, Z 385.949, A -106.87, B 85.042, C -82.235, E1 0, E2 0, E3 0, E4 0}
LIN {X 556.655, Y 262.938, Z 385.918, A -106.87, B 85.042, C -82.235, E1 0, E2 0, E3 0, E4 0}
LIN {X 556.364, Y 264.172, Z 385.823, A -106.87, B 85.042, C -82.235, E1 0, E2 0, E3 0, E4 0}
LIN {X 558.263, Y 267.821, Z 385.473, A -106.87, B 85.042, C -82.235, E1 0, E2 0, E3 0, E4 0}
LIN {X 558.21, Y 271.549, Z 385.164, A -106.87, B 85.042, C -82.235, E1 0, E2 0, E3 0, E4 0}
LIN {X 558.501, Y 275.574, Z 384.823, A -106.87, B 85.042, C -82.235, E1 0, E2 0, E3 0, E4 0}
LIN {X 560.138, Y 308.411, Z 382.056, A -106.87, B 85.042, C -82.235, E1 0, E2 0, E3 0, E4 0}
LIN {X 559.783, Y 313.294, Z 381.659, A -106.87, B 85.042, C -82.235, E1 0, E2 0, E3 0, E4 0}
LIN {X 560.181, Y 314.89, Z 381.516, A -106.87, B 85.042, C -82.235, E1 0, E2 0, E3 0, E4 0}
LIN {X 560.098, Y 315.919, Z 381.433, A -106.87, B 85.042, C -82.235, E1 0, E2 0, E3 0, E4 0}
LIN {X 560.064, Y 315.988, Z 381.428, A -106.87, B 85.042, C -82.235, E1 0, E2 0, E3 0, E4 0}
LIN {X 560.432, Y 329.432, Z 380.303, A -106.87, B 85.042, C -82.235, E1 0, E2 0, E3 0, E4 0}
LIN {X 560.356, Y 329.592, Z 380.292, A -106.87, B 85.042, C -82.235, E1 0, E2 0, E3 0, E4 0}
LIN {X 559.41, Y 334.898, Z 379.875, A -106.87, B 85.042, C -82.235, E1 0, E2 0, E3 0, E4 0}
LIN {X 559.482, Y 349.609, Z 378.652, A -106.87, B 85.042, C -82.235, E1 0, E2 0, E3 0, E4 0}
LIN {X 559.544, Y 351.384, Z 378.503, A -106.87, B 85.042, C -82.235, E1 0, E2 0, E3 0, E4 0}
LIN {X 578.308, Y 345.308, Z 378.535, A -106.87, B 85.042, C -82.235, E1 0, E2 0, E3 0, E4 0}
LIN {X 593.592, Y 343.953, Z 378.263, A -106.87, B 85.042, C -82.235, E1 0, E2 0, E3 0, E4 0}
LIN {X 593.538, Y 343.773, Z 376.097, A -106.87, B 85.042, C -82.235, E1 0, E2 0, E3 0, E4 0}
LIN {X 595.101, Y 343.057, Z 376.117, A -106.87, B 85.042, C -82.235, E1 0, E2 0, E3 0, E4 0}
LIN {X 597.129, Y 336.649, Z 376.598, A -106.87, B 85.042, C -82.235, E1 0, E2 0, E3 0, E4 0}
LIN {X 575.756, Y 346.437, Z 376.323, A -106.87, B 85.042, C -82.235, E1 0, E2 0, E3 0, E4 0}
LIN {X 559.438, Y 348.431, Z 376.569, A -106.87, B 85.042, C -82.235, E1 0, E2 0, E3 0, E4 0}
LIN {X 594.994, Y 332.148, Z 377.025, A -106.87, B 85.042, C -82.235, E1 0, E2 0, E3 0, E4 0}
LIN {X 593.053, Y 327.558, Z 377.455, A -106.87, B 85.042, C -82.235, E1 0, E2 0, E3 0, E4 0}
LIN {X 559.319, Y 343.006, Z 377.022, A -106.87, B 85.042, C -82.235, E1 0, E2 0, E3 0, E4 0}
LIN {X 559.261, Y 337.554, Z 377.476, A -106.87, B 85.042, C -82.235, E1 0, E2 0, E3 0, E4 0}
LIN {X 591.34, Y 322.863, Z 377.888, A -106.87, B 85.042, C -82.235, E1 0, E2 0, E3 0, E4 0}
LIN {X 588.924, Y 318.49, Z 378.312, A -106.87, B 85.042, C -82.235, E1 0, E2 0, E3 0, E4 0}
LIN {X 560.003, Y 331.735, Z 377.941, A -106.87, B 85.042, C -82.235, E1 0, E2 0, E3 0, E4 0}
LIN {X 560.118, Y 326.203, Z 378.397, A -106.87, B 85.042, C -82.235, E1 0, E2 0, E3 0, E4 0}
LIN {X 586.732, Y 314.015, Z 378.739, A -106.87, B 85.042, C -82.235, E1 0, E2 0, E3 0, E4 0}
LIN {X 584.695, Y 309.468, Z 379.168, A -106.87, B 85.042, C -82.235, E1 0, E2 0, E3 0, E4 0}
LIN {X 559.941, Y 320.805, Z 378.849, A -106.87, B 85.042, C -82.235, E1 0, E2 0, E3 0, E4 0}
LIN {X 560.058, Y 315.272, Z 379.306, A -106.87, B 85.042, C -82.235, E1 0, E2 0, E3 0, E4 0}
LIN {X 582.628, Y 304.936, Z 379.596, A -106.87, B 85.042, C -82.235, E1 0, E2 0, E3 0, E4 0}
LIN {X 580.672, Y 300.352, Z 380.026, A -106.87, B 85.042, C -82.235, E1 0, E2 0, E3 0, E4 0}
LIN {X 560.024, Y 309.808, Z 379.76, A -106.87, B 85.042, C -82.235, E1 0, E2 0, E3 0, E4 0}
LIN {X 559.741, Y 304.459, Z 380.211, A -106.87, B 85.042, C -82.235, E1 0, E2 0, E3 0, E4 0}
LIN {X 578.868, Y 295.699, Z 380.457, A -106.87, B 85.042, C -82.235, E1 0, E2 0, E3 0, E4 0}
LIN {X 576.955, Y 291.097, Z 380.888, A -106.87, B 85.042, C -82.235, E1 0, E2 0, E3 0, E4 0}
LIN {X 559.489, Y 299.095, Z 380.663, A -106.87, B 85.042, C -82.235, E1 0, E2 0, E3 0, E4 0}
LIN {X 559.694, Y 293.522, Z 381.121, A -106.87, B 85.042, C -82.235, E1 0, E2 0, E3 0, E4 0}
LIN {X 575.244, Y 286.401, Z 381.32, A -106.87, B 85.042, C -82.235, E1 0, E2 0, E3 0, E4 0}
LIN {X 573.234, Y 281.842, Z 381.749, A -106.87, B 85.042, C -82.235, E1 0, E2 0, E3 0, E4 0}
LIN {X 559.282, Y 288.232, Z 381.57, A -106.87, B 85.042, C -82.235, E1 0, E2 0, E3 0, E4 0}
LIN {X 558.624, Y 283.054, Z 382.017, A -106.87, B 85.042, C -82.235, E1 0, E2 0, E3 0, E4 0}
LIN {X 571.262, Y 277.266, Z 382.179, A -106.87, B 85.042, C -82.235, E1 0, E2 0, E3 0, E4 0}
LIN {X 569.124, Y 272.766, Z 382.607, A -106.87, B 85.042, C -82.235, E1 0, E2 0, E3 0, E4 0}
LIN {X 558.462, Y 277.649, Z 382.47, A -106.87, B 85.042, C -82.235, E1 0, E2 0, E3 0, E4 0}
LIN {X 558.136, Y 272.319, Z 382.92, A -106.87, B 85.042, C -82.235, E1 0, E2 0, E3 0, E4 0}
LIN {X 567.243, Y 268.148, Z 383.037, A -106.87, B 85.042, C -82.235, E1 0, E2 0, E3 0, E4 0}
LIN {X 565.487, Y 263.473, Z 383.47, A -106.87, B 85.042, C -82.235, E1 0, E2 0, E3 0, E4 0}
LIN {X 557.997, Y 266.904, Z 383.373, A -106.87, B 85.042, C -82.235, E1 0, E2 0, E3 0, E4 0}
LIN {X 578.659, Y 345.787, Z 376.304, A -106.87, B 85.042, C -82.235, E1 0, E2 0, E3 0, E4 0}
LIN {X 579.8, Y 345.087, Z 376.334, A -106.87, B 85.042, C -82.235, E1 0, E2 0, E3 0, E4 0}
LIN {X 586.254, Y 342.433, Z 376.391, A -106.87, B 85.042, C -82.235, E1 0, E2 0, E3 0, E4 0}
LIN {X 589.339, Y 342.295, Z 376.325, A -106.87, B 85.042, C -82.235, E1 0, E2 0, E3 0, E4 0}
LIN {X 591.467, Y 343.446, Z 376.176, A -106.87, B 85.042, C -82.235, E1 0, E2 0, E3 0, E4 0}
LIN {X 594.417, Y 344.016, Z 376.055, A -106.87, B 85.042, C -82.235, E1 0, E2 0, E3 0, E4 0}
LIN {X 594.909, Y 343.716, Z 376.067, A -106.87, B 85.042, C -82.235, E1 0, E2 0, E3 0, E4 0}
LIN {X 595.343, Y 342.449, Z 376.161, A -106.87, B 85.042, C -82.235, E1 0, E2 0, E3 0, E4 0}
LIN {X 595.416, Y 342.378, Z 376.165, A -106.87, B 85.042, C -82.235, E1 0, E2 0, E3 0, E4 0}
LIN {X 596.193, Y 340.567, Z 376.296, A -106.87, B 85.042, C -82.235, E1 0, E2 0, E3 0, E4 0}
LIN {X 597.689, Y 339.439, Z 376.352, A -106.87, B 85.042, C -82.235, E1 0, E2 0, E3 0, E4 0}
LIN {X 597.729, Y 339.003, Z 376.387, A -106.87, B 85.042, C -82.235, E1 0, E2 0, E3 0, E4 0}
LIN {X 597.471, Y 338.592, Z 376.428, A -106.87, B 85.042, C -82.235, E1 0, E2 0, E3 0, E4 0}
LIN {X 597.346, Y 337.075, Z 376.557, A -106.87, B 85.042, C -82.235, E1 0, E2 0, E3 0, E4 0}
LIN {X 594.421, Y 330.871, Z 377.146, A -106.87, B 85.042, C -82.235, E1 0, E2 0, E3 0, E4 0}
LIN {X 593.658, Y 330.04, Z 377.234, A -106.87, B 85.042, C -82.235, E1 0, E2 0, E3 0, E4 0}
LIN {X 591.059, Y 322.276, Z 377.944, A -106.87, B 85.042, C -82.235, E1 0, E2 0, E3 0, E4 0}
LIN {X 590.449, Y 321.533, Z 378.021, A -106.87, B 85.042, C -82.235, E1 0, E2 0, E3 0, E4 0}
LIN {X 590.093, Y 321.321, Z 378.048, A -106.87, B 85.042, C -82.235, E1 0, E2 0, E3 0, E4 0}
LIN {X 590.055, Y 321.363, Z 378.045, A -106.87, B 85.042, C -82.235, E1 0, E2 0, E3 0, E4 0}
LIN {X 589.83, Y 321.122, Z 378.071, A -106.87, B 85.042, C -82.235, E1 0, E2 0, E3 0, E4 0}
LIN {X 589.166, Y 319.351, Z 378.234, A -106.87, B 85.042, C -82.235, E1 0, E2 0, E3 0, E4 0}
LIN {X 589.115, Y 319.263, Z 378.243, A -106.87, B 85.042, C -82.235, E1 0, E2 0, E3 0, E4 0}
LIN {X 588.865, Y 318.25, Z 378.333, A -106.87, B 85.042, C -82.235, E1 0, E2 0, E3 0, E4 0}
LIN {X 588.294, Y 317.474, Z 378.412, A -106.87, B 85.042, C -82.235, E1 0, E2 0, E3 0, E4 0}
LIN {X 588.047, Y 316.503, Z 378.499, A -106.87, B 85.042, C -82.235, E1 0, E2 0, E3 0, E4 0}
LIN {X 587.451, Y 315.728, Z 378.578, A -106.87, B 85.042, C -82.235, E1 0, E2 0, E3 0, E4 0}
LIN {X 587.474, Y 315.405, Z 378.605, A -106.87, B 85.042, C -82.235, E1 0, E2 0, E3 0, E4 0}
LIN {X 586.501, Y 313.669, Z 378.773, A -106.87, B 85.042, C -82.235, E1 0, E2 0, E3 0, E4 0}
LIN {X 586.305, Y 312.469, Z 378.878, A -106.87, B 85.042, C -82.235, E1 0, E2 0, E3 0, E4 0}
LIN {X 585.166, Y 310.311, Z 379.086, A -106.87, B 85.042, C -82.235, E1 0, E2 0, E3 0, E4 0}
LIN {X 584.808, Y 309.964, Z 379.124, A -106.87, B 85.042, C -82.235, E1 0, E2 0, E3 0, E4 0}
LIN {X 584.153, Y 307.357, Z 379.356, A -106.87, B 85.042, C -82.235, E1 0, E2 0, E3 0, E4 0}
LIN {X 582.178, Y 304.32, Z 379.658, A -106.87, B 85.042, C -82.235, E1 0, E2 0, E3 0, E4 0}
LIN {X 582.171, Y 304.28, Z 379.662, A -106.87, B 85.042, C -82.235, E1 0, E2 0, E3 0, E4 0}
LIN {X 581.578, Y 303.354, Z 379.754, A -106.87, B 85.042, C -82.235, E1 0, E2 0, E3 0, E4 0}
LIN {X 581.051, Y 301.368, Z 379.932, A -106.87, B 85.042, C -82.235, E1 0, E2 0, E3 0, E4 0}
LIN {X 581.008, Y 301.307, Z 379.938, A -106.87, B 85.042, C -82.235, E1 0, E2 0, E3 0, E4 0}
LIN {X 580.4, Y 299.159, Z 380.131, A -106.87, B 85.042, C -82.235, E1 0, E2 0, E3 0, E4 0}
LIN {X 564.652, Y 261.251, Z 383.675, A -106.87, B 85.042, C -82.235, E1 0, E2 0, E3 0, E4 0}
LIN {X 562.815, Y 261.737, Z 383.681, A -106.87, B 85.042, C -82.235, E1 0, E2 0, E3 0, E4 0}
LIN {X 562.777, Y 261.804, Z 383.676, A -106.87, B 85.042, C -82.235, E1 0, E2 0, E3 0, E4 0}
LIN {X 561.986, Y 261.957, Z 383.683, A -106.87, B 85.042, C -82.235, E1 0, E2 0, E3 0, E4 0}
LIN {X 561.537, Y 261.894, Z 383.7, A -106.87, B 85.042, C -82.235, E1 0, E2 0, E3 0, E4 0}
LIN {X 561.504, Y 261.78, Z 383.71, A -106.87, B 85.042, C -82.235, E1 0, E2 0, E3 0, E4 0}
LIN {X 560.1, Y 261.485, Z 383.77, A -106.87, B 85.042, C -82.235, E1 0, E2 0, E3 0, E4 0}
LIN {X 557.658, Y 262.243, Z 383.769, A -106.87, B 85.042, C -82.235, E1 0, E2 0, E3 0, E4 0}
LIN {X 557.037, Y 262.254, Z 383.783, A -106.87, B 85.042, C -82.235, E1 0, E2 0, E3 0, E4 0}
LIN {X 556.601, Y 262.758, Z 383.753, A -106.87, B 85.042, C -82.235, E1 0, E2 0, E3 0, E4 0}
LIN {X 556.31, Y 263.993, Z 383.657, A -106.87, B 85.042, C -82.235, E1 0, E2 0, E3 0, E4 0}
LIN {X 558.209, Y 267.641, Z 383.307, A -106.87, B 85.042, C -82.235, E1 0, E2 0, E3 0, E4 0}
LIN {X 558.155, Y 271.369, Z 382.999, A -106.87, B 85.042, C -82.235, E1 0, E2 0, E3 0, E4 0}
LIN {X 558.447, Y 275.394, Z 382.657, A -106.87, B 85.042, C -82.235, E1 0, E2 0, E3 0, E4 0}
LIN {X 560.083, Y 308.231, Z 379.89, A -106.87, B 85.042, C -82.235, E1 0, E2 0, E3 0, E4 0}
LIN {X 559.729, Y 313.114, Z 379.493, A -106.87, B 85.042, C -82.235, E1 0, E2 0, E3 0, E4 0}
LIN {X 560.126, Y 314.711, Z 379.351, A -106.87, B 85.042, C -82.235, E1 0, E2 0, E3 0, E4 0}
LIN {X 560.044, Y 315.74, Z 379.267, A -106.87, B 85.042, C -82.235, E1 0, E2 0, E3 0, E4 0}
LIN {X 560.009, Y 315.808, Z 379.262, A -106.87, B 85.042, C -82.235, E1 0, E2 0, E3 0, E4 0}
LIN {X 560.378, Y 329.253, Z 378.137, A -106.87, B 85.042, C -82.235, E1 0, E2 0, E3 0, E4 0}
LIN {X 560.301, Y 329.413, Z 378.126, A -106.87, B 85.042, C -82.235, E1 0, E2 0, E3 0, E4 0}
LIN {X 559.355, Y 334.718, Z 377.709, A -106.87, B 85.042, C -82.235, E1 0, E2 0, E3 0, E4 0}
LIN {X 559.527, Y 346.823, Z 376.7, A -106.87, B 85.042, C -82.235, E1 0, E2 0, E3 0, E4 0}
LIN {X 559.454, Y 347.081, Z 376.68, A -106.87, B 85.042, C -82.235, E1 0, E2 0, E3 0, E4 0}
LIN {X 559.497, Y 351.75, Z 376.292, A -106.87, B 85.042, C -82.235, E1 0, E2 0, E3 0, E4 0}
LIN {X 559.55, Y 352.22, Z 376.251, A -106.87, B 85.042, C -82.235, E1 0, E2 0, E3 0, E4 0}
LIN {X 560.362, Y 351.97, Z 376.251, A -106.87, B 85.042, C -82.235, E1 0, E2 0, E3 0, E4 0}
LIN {X 562.452, Y 350.388, Z 376.33, A -106.87, B 85.042, C -82.235, E1 0, E2 0, E3 0, E4 0}
LIN {X 565.785, Y 349.073, Z 376.356, A -106.87, B 85.042, C -82.235, E1 0, E2 0, E3 0, E4 0}
LIN {X 574.203, Y 346.589, Z 376.35, A -106.87, B 85.042, C -82.235, E1 0, E2 0, E3 0, E4 0}
LIN {X 574.84, Y 346.246, Z 376.362, A -106.87, B 85.042, C -82.235, E1 0, E2 0, E3 0, E4 0}
LIN {X 576.319, Y 346.566, Z 376.299, A -106.87, B 85.042, C -82.235, E1 0, E2 0, E3 0, E4 0}
LIN {X 577.779, Y 346.327, Z 376.282, A -106.87, B 85.042, C -82.235, E1 0, E2 0, E3 0, E4 0}
LIN {X 578.659, Y 345.787, Z 376.304, A -106.87, B 85.042, C -82.235, E1 0, E2 0, E3 0, E4 0}
LIN {X 597.335, Y 336.555, Z 376.601, A -106.87, B 85.042, C -82.235, E1 0, E2 0, E3 0, E4 0}
LIN {X 597.281, Y 336.375, Z 374.435, A -106.87, B 85.042, C -82.235, E1 0, E2 0, E3 0, E4 0}
LIN {X 576.023, Y 346.111, Z 374.162, A -106.87, B 85.042, C -82.235, E1 0, E2 0, E3 0, E4 0}
LIN {X 559.383, Y 348.252, Z 374.403, A -106.87, B 85.042, C -82.235, E1 0, E2 0, E3 0, E4 0}
LIN {X 595.116, Y 331.887, Z 374.862, A -106.87, B 85.042, C -82.235, E1 0, E2 0, E3 0, E4 0}
LIN {X 593.132, Y 327.317, Z 375.291, A -106.87, B 85.042, C -82.235, E1 0, E2 0, E3 0, E4 0}
LIN {X 559.265, Y 342.827, Z 374.856, A -106.87, B 85.042, C -82.235, E1 0, E2 0, E3 0, E4 0}
LIN {X 559.207, Y 337.374, Z 375.31, A -106.87, B 85.042, C -82.235, E1 0, E2 0, E3 0, E4 0}
LIN {X 591.33, Y 322.663, Z 375.723, A -106.87, B 85.042, C -82.235, E1 0, E2 0, E3 0, E4 0}
LIN {X 589.115, Y 318.198, Z 376.149, A -106.87, B 85.042, C -82.235, E1 0, E2 0, E3 0, E4 0}
LIN {X 559.948, Y 331.555, Z 375.775, A -106.87, B 85.042, C -82.235, E1 0, E2 0, E3 0, E4 0}
LIN {X 560.063, Y 326.023, Z 376.231, A -106.87, B 85.042, C -82.235, E1 0, E2 0, E3 0, E4 0}
LIN {X 586.862, Y 313.751, Z 376.575, A -106.87, B 85.042, C -82.235, E1 0, E2 0, E3 0, E4 0}
LIN {X 585.185, Y 309.039, Z 377.009, A -106.87, B 85.042, C -82.235, E1 0, E2 0, E3 0, E4 0}
LIN {X 559.887, Y 320.625, Z 376.684, A -106.87, B 85.042, C -82.235, E1 0, E2 0, E3 0, E4 0}
LIN {X 560.004, Y 315.092, Z 377.14, A -106.87, B 85.042, C -82.235, E1 0, E2 0, E3 0, E4 0}
LIN {X 582.993, Y 304.564, Z 377.435, A -106.87, B 85.042, C -82.235, E1 0, E2 0, E3 0, E4 0}
LIN {X 581.23, Y 299.892, Z 377.867, A -106.87, B 85.042, C -82.235, E1 0, E2 0, E3 0, E4 0}
LIN {X 559.97, Y 309.629, Z 377.594, A -106.87, B 85.042, C -82.235, E1 0, E2 0, E3 0, E4 0}
LIN {X 559.686, Y 304.279, Z 378.046, A -106.87, B 85.042, C -82.235, E1 0, E2 0, E3 0, E4 0}
LIN {X 579.248, Y 295.321, Z 378.297, A -106.87, B 85.042, C -82.235, E1 0, E2 0, E3 0, E4 0}
LIN {X 577.025, Y 290.86, Z 378.723, A -106.87, B 85.042, C -82.235, E1 0, E2 0, E3 0, E4 0}
LIN {X 559.435, Y 298.915, Z 378.497, A -106.87, B 85.042, C -82.235, E1 0, E2 0, E3 0, E4 0}
LIN {X 559.64, Y 293.342, Z 378.955, A -106.87, B 85.042, C -82.235, E1 0, E2 0, E3 0, E4 0}
LIN {X 575.327, Y 286.158, Z 379.156, A -106.87, B 85.042, C -82.235, E1 0, E2 0, E3 0, E4 0}
LIN {X 573.429, Y 281.548, Z 379.587, A -106.87, B 85.042, C -82.235, E1 0, E2 0, E3 0, E4 0}
LIN {X 559.228, Y 288.052, Z 379.405, A -106.87, B 85.042, C -82.235, E1 0, E2 0, E3 0, E4 0}
LIN {X 558.569, Y 282.874, Z 379.851, A -106.87, B 85.042, C -82.235, E1 0, E2 0, E3 0, E4 0}
LIN {X 571.858, Y 276.788, Z 380.022, A -106.87, B 85.042, C -82.235, E1 0, E2 0, E3 0, E4 0}
LIN {X 569.28, Y 272.49, Z 380.443, A -106.87, B 85.042, C -82.235, E1 0, E2 0, E3 0, E4 0}
LIN {X 558.408, Y 277.469, Z 380.304, A -106.87, B 85.042, C -82.235, E1 0, E2 0, E3 0, E4 0}
LIN {X 558.082, Y 272.139, Z 380.754, A -106.87, B 85.042, C -82.235, E1 0, E2 0, E3 0, E4 0}
LIN {X 567.429, Y 267.858, Z 380.875, A -106.87, B 85.042, C -82.235, E1 0, E2 0, E3 0, E4 0}
LIN {X 565.675, Y 263.182, Z 381.307, A -106.87, B 85.042, C -82.235, E1 0, E2 0, E3 0, E4 0}
LIN {X 557.942, Y 266.724, Z 381.208, A -106.87, B 85.042, C -82.235, E1 0, E2 0, E3 0, E4 0}
LIN {X 578.608, Y 345.621, Z 374.137, A -106.87, B 85.042, C -82.235, E1 0, E2 0, E3 0, E4 0}
LIN {X 579.018, Y 345.535, Z 374.134, A -106.87, B 85.042, C -82.235, E1 0, E2 0, E3 0, E4 0}
LIN {X 586.169, Y 342.8, Z 374.181, A -106.87, B 85.042, C -82.235, E1 0, E2 0, E3 0, E4 0}
LIN {X 593.35, Y 342.74, Z 374.005, A -106.87, B 85.042, C -82.235, E1 0, E2 0, E3 0, E4 0}
LIN {X 594.096, Y 342.472, Z 374.009, A -106.87, B 85.042, C -82.235, E1 0, E2 0, E3 0, E4 0}
LIN {X 596.271, Y 340.714, Z 374.1, A -106.87, B 85.042, C -82.235, E1 0, E2 0, E3 0, E4 0}
LIN {X 596.544, Y 340.212, Z 374.135, A -106.87, B 85.042, C -82.235, E1 0, E2 0, E3 0, E4 0}
LIN {X 597.229, Y 339.555, Z 374.172, A -106.87, B 85.042, C -82.235, E1 0, E2 0, E3 0, E4 0}
LIN {X 598.01, Y 339.356, Z 374.169, A -106.87, B 85.042, C -82.235, E1 0, E2 0, E3 0, E4 0}
LIN {X 598.257, Y 338.761, Z 374.212, A -106.87, B 85.042, C -82.235, E1 0, E2 0, E3 0, E4 0}
LIN {X 598.278, Y 338.738, Z 374.213, A -106.87, B 85.042, C -82.235, E1 0, E2 0, E3 0, E4 0}
LIN {X 598.099, Y 338.067, Z 374.274, A -106.87, B 85.042, C -82.235, E1 0, E2 0, E3 0, E4 0}
LIN {X 597.454, Y 337.262, Z 374.357, A -106.87, B 85.042, C -82.235, E1 0, E2 0, E3 0, E4 0}
LIN {X 597.351, Y 337.048, Z 374.377, A -106.87, B 85.042, C -82.235, E1 0, E2 0, E3 0, E4 0}
LIN {X 597.236, Y 336.129, Z 374.456, A -106.87, B 85.042, C -82.235, E1 0, E2 0, E3 0, E4 0}
LIN {X 596.555, Y 334.793, Z 374.584, A -106.87, B 85.042, C -82.235, E1 0, E2 0, E3 0, E4 0}
LIN {X 596.294, Y 334.585, Z 374.608, A -106.87, B 85.042, C -82.235, E1 0, E2 0, E3 0, E4 0}
LIN {X 595.928, Y 333.759, Z 374.686, A -106.87, B 85.042, C -82.235, E1 0, E2 0, E3 0, E4 0}
LIN {X 595.873, Y 333.707, Z 374.692, A -106.87, B 85.042, C -82.235, E1 0, E2 0, E3 0, E4 0}
LIN {X 593.176, Y 327.766, Z 375.253, A -106.87, B 85.042, C -82.235, E1 0, E2 0, E3 0, E4 0}
LIN {X 593.069, Y 326.599, Z 375.352, A -106.87, B 85.042, C -82.235, E1 0, E2 0, E3 0, E4 0}
LIN {X 591.325, Y 322.655, Z 375.724, A -106.87, B 85.042, C -82.235, E1 0, E2 0, E3 0, E4 0}
LIN {X 591.116, Y 321.864, Z 375.795, A -106.87, B 85.042, C -82.235, E1 0, E2 0, E3 0, E4 0}
LIN {X 590.969, Y 321.693, Z 375.813, A -106.87, B 85.042, C -82.235, E1 0, E2 0, E3 0, E4 0}
LIN {X 585.269, Y 309.25, Z 376.989, A -106.87, B 85.042, C -82.235, E1 0, E2 0, E3 0, E4 0}
LIN {X 582.379, Y 303.657, Z 377.526, A -106.87, B 85.042, C -82.235, E1 0, E2 0, E3 0, E4 0}
LIN {X 575.336, Y 286.254, Z 379.148, A -106.87, B 85.042, C -82.235, E1 0, E2 0, E3 0, E4 0}
LIN {X 575.266, Y 285.509, Z 379.212, A -106.87, B 85.042, C -82.235, E1 0, E2 0, E3 0, E4 0}
LIN {X 571.833, Y 276.704, Z 380.029, A -106.87, B 85.042, C -82.235, E1 0, E2 0, E3 0, E4 0}
LIN {X 570.894, Y 275.716, Z 380.135, A -106.87, B 85.042, C -82.235, E1 0, E2 0, E3 0, E4 0}
LIN {X 564.885, Y 260.991, Z 381.509, A -106.87, B 85.042, C -82.235, E1 0, E2 0, E3 0, E4 0}
LIN {X 562.76, Y 261.557, Z 381.515, A -106.87, B 85.042, C -82.235, E1 0, E2 0, E3 0, E4 0}
LIN {X 562.723, Y 261.624, Z 381.511, A -106.87, B 85.042, C -82.235, E1 0, E2 0, E3 0, E4 0}
LIN {X 561.931, Y 261.777, Z 381.518, A -106.87, B 85.042, C -82.235, E1 0, E2 0, E3 0, E4 0}
LIN {X 561.482, Y 261.714, Z 381.534, A -106.87, B 85.042, C -82.235, E1 0, E2 0, E3 0, E4 0}
LIN {X 561.449, Y 261.601, Z 381.544, A -106.87, B 85.042, C -82.235, E1 0, E2 0, E3 0, E4 0}
LIN {X 560.046, Y 261.305, Z 381.604, A -106.87, B 85.042, C -82.235, E1 0, E2 0, E3 0, E4 0}
LIN {X 557.603, Y 262.063, Z 381.603, A -106.87, B 85.042, C -82.235, E1 0, E2 0, E3 0, E4 0}
LIN {X 556.982, Y 262.074, Z 381.618, A -106.87, B 85.042, C -82.235, E1 0, E2 0, E3 0, E4 0}
LIN {X 556.546, Y 262.578, Z 381.587, A -106.87, B 85.042, C -82.235, E1 0, E2 0, E3 0, E4 0}
LIN {X 556.255, Y 263.813, Z 381.492, A -106.87, B 85.042, C -82.235, E1 0, E2 0, E3 0, E4 0}
LIN {X 558.154, Y 267.461, Z 381.141, A -106.87, B 85.042, C -82.235, E1 0, E2 0, E3 0, E4 0}
LIN {X 558.101, Y 271.189, Z 380.833, A -106.87, B 85.042, C -82.235, E1 0, E2 0, E3 0, E4 0}
LIN {X 558.392, Y 275.214, Z 380.491, A -106.87, B 85.042, C -82.235, E1 0, E2 0, E3 0, E4 0}
LIN {X 560.029, Y 308.052, Z 377.724, A -106.87, B 85.042, C -82.235, E1 0, E2 0, E3 0, E4 0}
LIN {X 559.674, Y 312.934, Z 377.328, A -106.87, B 85.042, C -82.235, E1 0, E2 0, E3 0, E4 0}
LIN {X 560.072, Y 314.531, Z 377.185, A -106.87, B 85.042, C -82.235, E1 0, E2 0, E3 0, E4 0}
LIN {X 559.989, Y 315.56, Z 377.102, A -106.87, B 85.042, C -82.235, E1 0, E2 0, E3 0, E4 0}
LIN {X 559.955, Y 315.628, Z 377.097, A -106.87, B 85.042, C -82.235, E1 0, E2 0, E3 0, E4 0}
LIN {X 560.323, Y 329.073, Z 375.971, A -106.87, B 85.042, C -82.235, E1 0, E2 0, E3 0, E4 0}
LIN {X 560.247, Y 329.233, Z 375.96, A -106.87, B 85.042, C -82.235, E1 0, E2 0, E3 0, E4 0}
LIN {X 559.301, Y 334.538, Z 375.543, A -106.87, B 85.042, C -82.235, E1 0, E2 0, E3 0, E4 0}
LIN {X 559.472, Y 346.644, Z 374.534, A -106.87, B 85.042, C -82.235, E1 0, E2 0, E3 0, E4 0}
LIN {X 559.4, Y 346.902, Z 374.514, A -106.87, B 85.042, C -82.235, E1 0, E2 0, E3 0, E4 0}
LIN {X 559.443, Y 351.571, Z 374.126, A -106.87, B 85.042, C -82.235, E1 0, E2 0, E3 0, E4 0}
LIN {X 559.535, Y 352.475, Z 374.048, A -106.87, B 85.042, C -82.235, E1 0, E2 0, E3 0, E4 0}
LIN {X 561.343, Y 352.31, Z 374.017, A -106.87, B 85.042, C -82.235, E1 0, E2 0, E3 0, E4 0}
LIN {X 567.584, Y 348.32, Z 374.191, A -106.87, B 85.042, C -82.235, E1 0, E2 0, E3 0, E4 0}
LIN {X 567.742, Y 348.062, Z 374.208, A -106.87, B 85.042, C -82.235, E1 0, E2 0, E3 0, E4 0}
LIN {X 568.615, Y 347.473, Z 374.235, A -106.87, B 85.042, C -82.235, E1 0, E2 0, E3 0, E4 0}
LIN {X 569.541, Y 347.212, Z 374.233, A -106.87, B 85.042, C -82.235, E1 0, E2 0, E3 0, E4 0}
LIN {X 571.244, Y 346.578, Z 374.243, A -106.87, B 85.042, C -82.235, E1 0, E2 0, E3 0, E4 0}
LIN {X 573.605, Y 345.996, Z 374.232, A -106.87, B 85.042, C -82.235, E1 0, E2 0, E3 0, E4 0}
LIN {X 576.191, Y 346.129, Z 374.156, A -106.87, B 85.042, C -82.235, E1 0, E2 0, E3 0, E4 0}
LIN {X 578.608, Y 345.621, Z 374.137, A -106.87, B 85.042, C -82.235, E1 0, E2 0, E3 0, E4 0}
LIN {X 597.587, Y 336.235, Z 374.439, A -106.87, B 85.042, C -82.235, E1 0, E2 0, E3 0, E4 0}
LIN {X 597.533, Y 336.055, Z 372.273, A -106.87, B 85.042, C -82.235, E1 0, E2 0, E3 0, E4 0}
LIN {X 576.509, Y 345.683, Z 372.003, A -106.87, B 85.042, C -82.235, E1 0, E2 0, E3 0, E4 0}
LIN {X 562.592, Y 352.056, Z 371.824, A -106.87, B 85.042, C -82.235, E1 0, E2 0, E3 0, E4 0}
LIN {X 568.057, Y 349.554, Z 371.894, A -106.87, B 85.042, C -82.235, E1 0, E2 0, E3 0, E4 0}
LIN {X 595.242, Y 331.625, Z 372.698, A -106.87, B 85.042, C -82.235, E1 0, E2 0, E3 0, E4 0}
LIN {X 559.329, Y 348.072, Z 372.237, A -106.87, B 85.042, C -82.235, E1 0, E2 0, E3 0, E4 0}
LIN {X 559.21, Y 342.647, Z 372.69, A -106.87, B 85.042, C -82.235, E1 0, E2 0, E3 0, E4 0}
LIN {X 593.379, Y 326.999, Z 373.129, A -106.87, B 85.042, C -82.235, E1 0, E2 0, E3 0, E4 0}
LIN {X 591.329, Y 322.458, Z 373.558, A -106.87, B 85.042, C -82.235, E1 0, E2 0, E3 0, E4 0}
LIN {X 559.152, Y 337.194, Z 373.145, A -106.87, B 85.042, C -82.235, E1 0, E2 0, E3 0, E4 0}
LIN {X 559.893, Y 331.375, Z 373.609, A -106.87, B 85.042, C -82.235, E1 0, E2 0, E3 0, E4 0}
LIN {X 589.22, Y 317.945, Z 373.986, A -106.87, B 85.042, C -82.235, E1 0, E2 0, E3 0, E4 0}
LIN {X 587.369, Y 313.314, Z 374.417, A -106.87, B 85.042, C -82.235, E1 0, E2 0, E3 0, E4 0}
LIN {X 560.009, Y 325.843, Z 374.065, A -106.87, B 85.042, C -82.235, E1 0, E2 0, E3 0, E4 0}
LIN {X 559.832, Y 320.445, Z 374.518, A -106.87, B 85.042, C -82.235, E1 0, E2 0, E3 0, E4 0}
